(* IEC 61131-3 sources: TA/Tests/RetainTest/OLD/Structure test (part 11) *)

    MATRIX_STRUCTURE_RETAIN.MATRIX_STRING[7,0] := MATRIX_STRUCTURE_RETAIN.MATRIX_STRING[6,0];
    MATRIX_STRUCTURE_RETAIN.MATRIX_STRING[7,1] := MATRIX_STRUCTURE_RETAIN.MATRIX_STRING[6,1];
    MATRIX_STRUCTURE_RETAIN.MATRIX_STRING[7,2] := MATRIX_STRUCTURE_RETAIN.MATRIX_STRING[6,2];
    MATRIX_STRUCTURE_RETAIN.MATRIX_STRING[7,3] := MATRIX_STRUCTURE_RETAIN.MATRIX_STRING[6,3];
    MATRIX_STRUCTURE_RETAIN.MATRIX_STRING[7,4] := MATRIX_STRUCTURE_RETAIN.MATRIX_STRING[6,4];
    MATRIX_STRUCTURE_RETAIN.MATRIX_STRING[7,5] := MATRIX_STRUCTURE_RETAIN.MATRIX_STRING[6,5];
    MATRIX_STRUCTURE_RETAIN.MATRIX_STRING[7,6] := MATRIX_STRUCTURE_RETAIN.MATRIX_STRING[6,6];
    MATRIX_STRUCTURE_RETAIN.MATRIX_STRING[7,7] := MATRIX_STRUCTURE_RETAIN.MATRIX_STRING[6,7];
    MATRIX_STRUCTURE_RETAIN.MATRIX_STRING[7,8] := MATRIX_STRUCTURE_RETAIN.MATRIX_STRING[6,8];
    MATRIX_STRUCTURE_RETAIN.MATRIX_STRING[7,9] := MATRIX_STRUCTURE_RETAIN.MATRIX_STRING[6,9];

    MATRIX_STRUCTURE_RETAIN.MATRIX_TIME[0,0] := MATRIX_STRUCTURE_RETAIN.MATRIX_TIME[0,0] + PULSE_TIME;
    MATRIX_STRUCTURE_RETAIN.MATRIX_TIME[0,1] := MATRIX_STRUCTURE_RETAIN.MATRIX_TIME[0,1] + PULSE_TIME;
    MATRIX_STRUCTURE_RETAIN.MATRIX_TIME[0,2] := MATRIX_STRUCTURE_RETAIN.MATRIX_TIME[0,2] + PULSE_TIME;
    MATRIX_STRUCTURE_RETAIN.MATRIX_TIME[0,3] := MATRIX_STRUCTURE_RETAIN.MATRIX_TIME[0,3] + PULSE_TIME;
    MATRIX_STRUCTURE_RETAIN.MATRIX_TIME[0,4] := MATRIX_STRUCTURE_RETAIN.MATRIX_TIME[0,4] + PULSE_TIME;
    MATRIX_STRUCTURE_RETAIN.MATRIX_TIME[0,5] := MATRIX_STRUCTURE_RETAIN.MATRIX_TIME[0,5] + PULSE_TIME;
    MATRIX_STRUCTURE_RETAIN.MATRIX_TIME[0,6] := MATRIX_STRUCTURE_RETAIN.MATRIX_TIME[0,6] + PULSE_TIME;
    MATRIX_STRUCTURE_RETAIN.MATRIX_TIME[0,7] := MATRIX_STRUCTURE_RETAIN.MATRIX_TIME[0,7] + PULSE_TIME;
    MATRIX_STRUCTURE_RETAIN.MATRIX_TIME[0,8] := MATRIX_STRUCTURE_RETAIN.MATRIX_TIME[0,6];
    MATRIX_STRUCTURE_RETAIN.MATRIX_TIME[0,9] := MATRIX_STRUCTURE_RETAIN.MATRIX_TIME[0,7];

    MATRIX_STRUCTURE_RETAIN.MATRIX_TIME[1,0] := MATRIX_STRUCTURE_RETAIN.MATRIX_TIME[1,0] + PULSE_TIME;
    MATRIX_STRUCTURE_RETAIN.MATRIX_TIME[1,1] := MATRIX_STRUCTURE_RETAIN.MATRIX_TIME[1,1] + PULSE_TIME;
    MATRIX_STRUCTURE_RETAIN.MATRIX_TIME[1,2] := MATRIX_STRUCTURE_RETAIN.MATRIX_TIME[1,2] + PULSE_TIME;
    MATRIX_STRUCTURE_RETAIN.MATRIX_TIME[1,3] := MATRIX_STRUCTURE_RETAIN.MATRIX_TIME[1,3] + PULSE_TIME;
    MATRIX_STRUCTURE_RETAIN.MATRIX_TIME[1,4] := MATRIX_STRUCTURE_RETAIN.MATRIX_TIME[1,4] + PULSE_TIME;
    MATRIX_STRUCTURE_RETAIN.MATRIX_TIME[1,5] := MATRIX_STRUCTURE_RETAIN.MATRIX_TIME[1,5] + PULSE_TIME;
    MATRIX_STRUCTURE_RETAIN.MATRIX_TIME[1,6] := MATRIX_STRUCTURE_RETAIN.MATRIX_TIME[1,6] + PULSE_TIME;
    MATRIX_STRUCTURE_RETAIN.MATRIX_TIME[1,7] := MATRIX_STRUCTURE_RETAIN.MATRIX_TIME[1,7] + PULSE_TIME;
    MATRIX_STRUCTURE_RETAIN.MATRIX_TIME[1,8] := MATRIX_STRUCTURE_RETAIN.MATRIX_TIME[1,6];
    MATRIX_STRUCTURE_RETAIN.MATRIX_TIME[1,9] := MATRIX_STRUCTURE_RETAIN.MATRIX_TIME[1,7];

    MATRIX_STRUCTURE_RETAIN.MATRIX_TIME[2,0] := MATRIX_STRUCTURE_RETAIN.MATRIX_TIME[2,0] + PULSE_TIME;
    MATRIX_STRUCTURE_RETAIN.MATRIX_TIME[2,1] := MATRIX_STRUCTURE_RETAIN.MATRIX_TIME[2,1] + PULSE_TIME;
    MATRIX_STRUCTURE_RETAIN.MATRIX_TIME[2,2] := MATRIX_STRUCTURE_RETAIN.MATRIX_TIME[2,2] + PULSE_TIME;
    MATRIX_STRUCTURE_RETAIN.MATRIX_TIME[2,3] := MATRIX_STRUCTURE_RETAIN.MATRIX_TIME[2,3] + PULSE_TIME;
    MATRIX_STRUCTURE_RETAIN.MATRIX_TIME[2,4] := MATRIX_STRUCTURE_RETAIN.MATRIX_TIME[2,4] + PULSE_TIME;
    MATRIX_STRUCTURE_RETAIN.MATRIX_TIME[2,5] := MATRIX_STRUCTURE_RETAIN.MATRIX_TIME[2,5] + PULSE_TIME;
    MATRIX_STRUCTURE_RETAIN.MATRIX_TIME[2,6] := MATRIX_STRUCTURE_RETAIN.MATRIX_TIME[2,6] + PULSE_TIME;
    MATRIX_STRUCTURE_RETAIN.MATRIX_TIME[2,7] := MATRIX_STRUCTURE_RETAIN.MATRIX_TIME[2,7] + PULSE_TIME;
    MATRIX_STRUCTURE_RETAIN.MATRIX_TIME[2,8] := MATRIX_STRUCTURE_RETAIN.MATRIX_TIME[2,8] + PULSE_TIME;
    MATRIX_STRUCTURE_RETAIN.MATRIX_TIME[2,9] := MATRIX_STRUCTURE_RETAIN.MATRIX_TIME[2,9] + PULSE_TIME;

    MATRIX_STRUCTURE_RETAIN.MATRIX_TIME[3,0] := MATRIX_STRUCTURE_RETAIN.MATRIX_TIME[3,0] + PULSE_TIME;
    MATRIX_STRUCTURE_RETAIN.MATRIX_TIME[3,1] := MATRIX_STRUCTURE_RETAIN.MATRIX_TIME[3,1] + PULSE_TIME;
    MATRIX_STRUCTURE_RETAIN.MATRIX_TIME[3,2] := MATRIX_STRUCTURE_RETAIN.MATRIX_TIME[3,2] + PULSE_TIME;
    MATRIX_STRUCTURE_RETAIN.MATRIX_TIME[3,3] := MATRIX_STRUCTURE_RETAIN.MATRIX_TIME[3,3] + PULSE_TIME;
    MATRIX_STRUCTURE_RETAIN.MATRIX_TIME[3,4] := MATRIX_STRUCTURE_RETAIN.MATRIX_TIME[3,4] + PULSE_TIME;
    MATRIX_STRUCTURE_RETAIN.MATRIX_TIME[3,5] := MATRIX_STRUCTURE_RETAIN.MATRIX_TIME[3,5] + PULSE_TIME;
    MATRIX_STRUCTURE_RETAIN.MATRIX_TIME[3,6] := MATRIX_STRUCTURE_RETAIN.MATRIX_TIME[3,6] + PULSE_TIME;
    MATRIX_STRUCTURE_RETAIN.MATRIX_TIME[3,7] := MATRIX_STRUCTURE_RETAIN.MATRIX_TIME[3,7] + PULSE_TIME;
    MATRIX_STRUCTURE_RETAIN.MATRIX_TIME[3,8] := MATRIX_STRUCTURE_RETAIN.MATRIX_TIME[3,8] + PULSE_TIME;
    MATRIX_STRUCTURE_RETAIN.MATRIX_TIME[3,9] := MATRIX_STRUCTURE_RETAIN.MATRIX_TIME[3,9] + PULSE_TIME;

    MATRIX_STRUCTURE_RETAIN.MATRIX_TIME[4,0] := MATRIX_STRUCTURE_RETAIN.MATRIX_TIME[4,0] + PULSE_TIME;
    MATRIX_STRUCTURE_RETAIN.MATRIX_TIME[4,1] := MATRIX_STRUCTURE_RETAIN.MATRIX_TIME[4,1] + PULSE_TIME;
    MATRIX_STRUCTURE_RETAIN.MATRIX_TIME[4,2] := MATRIX_STRUCTURE_RETAIN.MATRIX_TIME[4,2] + PULSE_TIME;
    MATRIX_STRUCTURE_RETAIN.MATRIX_TIME[4,3] := MATRIX_STRUCTURE_RETAIN.MATRIX_TIME[4,3] + PULSE_TIME;
    MATRIX_STRUCTURE_RETAIN.MATRIX_TIME[4,4] := MATRIX_STRUCTURE_RETAIN.MATRIX_TIME[4,4] + PULSE_TIME;
    MATRIX_STRUCTURE_RETAIN.MATRIX_TIME[4,5] := MATRIX_STRUCTURE_RETAIN.MATRIX_TIME[4,5] + PULSE_TIME;
    MATRIX_STRUCTURE_RETAIN.MATRIX_TIME[4,6] := MATRIX_STRUCTURE_RETAIN.MATRIX_TIME[4,6] + PULSE_TIME;
    MATRIX_STRUCTURE_RETAIN.MATRIX_TIME[4,7] := MATRIX_STRUCTURE_RETAIN.MATRIX_TIME[4,7] + PULSE_TIME;
    MATRIX_STRUCTURE_RETAIN.MATRIX_TIME[4,8] := MATRIX_STRUCTURE_RETAIN.MATRIX_TIME[4,8] + PULSE_TIME;
    MATRIX_STRUCTURE_RETAIN.MATRIX_TIME[4,9] := MATRIX_STRUCTURE_RETAIN.MATRIX_TIME[4,9] + PULSE_TIME;

    MATRIX_STRUCTURE_RETAIN.MATRIX_TIME[5,0] := MATRIX_STRUCTURE_RETAIN.MATRIX_TIME[5,0] + PULSE_TIME;
    MATRIX_STRUCTURE_RETAIN.MATRIX_TIME[5,1] := MATRIX_STRUCTURE_RETAIN.MATRIX_TIME[5,1] + PULSE_TIME;
    MATRIX_STRUCTURE_RETAIN.MATRIX_TIME[5,2] := MATRIX_STRUCTURE_RETAIN.MATRIX_TIME[5,2] + PULSE_TIME;
    MATRIX_STRUCTURE_RETAIN.MATRIX_TIME[5,3] := MATRIX_STRUCTURE_RETAIN.MATRIX_TIME[5,3] + PULSE_TIME;
    MATRIX_STRUCTURE_RETAIN.MATRIX_TIME[5,4] := MATRIX_STRUCTURE_RETAIN.MATRIX_TIME[5,4] + PULSE_TIME;
    MATRIX_STRUCTURE_RETAIN.MATRIX_TIME[5,5] := MATRIX_STRUCTURE_RETAIN.MATRIX_TIME[5,5] + PULSE_TIME;
    MATRIX_STRUCTURE_RETAIN.MATRIX_TIME[5,6] := MATRIX_STRUCTURE_RETAIN.MATRIX_TIME[5,6] + PULSE_TIME;
    MATRIX_STRUCTURE_RETAIN.MATRIX_TIME[5,7] := MATRIX_STRUCTURE_RETAIN.MATRIX_TIME[5,7] + PULSE_TIME;
    MATRIX_STRUCTURE_RETAIN.MATRIX_TIME[5,8] := MATRIX_STRUCTURE_RETAIN.MATRIX_TIME[5,8] + PULSE_TIME;
    MATRIX_STRUCTURE_RETAIN.MATRIX_TIME[5,9] := MATRIX_STRUCTURE_RETAIN.MATRIX_TIME[5,9] + PULSE_TIME;

    MATRIX_STRUCTURE_RETAIN.MATRIX_TIME[6,0] := MATRIX_STRUCTURE_RETAIN.MATRIX_TIME[6,0] + PULSE_TIME;
    MATRIX_STRUCTURE_RETAIN.MATRIX_TIME[6,1] := MATRIX_STRUCTURE_RETAIN.MATRIX_TIME[6,1] + PULSE_TIME;
    MATRIX_STRUCTURE_RETAIN.MATRIX_TIME[6,2] := MATRIX_STRUCTURE_RETAIN.MATRIX_TIME[6,2] + PULSE_TIME;
    MATRIX_STRUCTURE_RETAIN.MATRIX_TIME[6,3] := MATRIX_STRUCTURE_RETAIN.MATRIX_TIME[6,3] + PULSE_TIME;
    MATRIX_STRUCTURE_RETAIN.MATRIX_TIME[6,4] := MATRIX_STRUCTURE_RETAIN.MATRIX_TIME[6,4] + PULSE_TIME;
    MATRIX_STRUCTURE_RETAIN.MATRIX_TIME[6,5] := MATRIX_STRUCTURE_RETAIN.MATRIX_TIME[6,5] + PULSE_TIME;
    MATRIX_STRUCTURE_RETAIN.MATRIX_TIME[6,6] := MATRIX_STRUCTURE_RETAIN.MATRIX_TIME[6,6] + PULSE_TIME;
    MATRIX_STRUCTURE_RETAIN.MATRIX_TIME[6,7] := MATRIX_STRUCTURE_RETAIN.MATRIX_TIME[6,7] + PULSE_TIME;
    MATRIX_STRUCTURE_RETAIN.MATRIX_TIME[6,8] := MATRIX_STRUCTURE_RETAIN.MATRIX_TIME[6,8] + PULSE_TIME;
    MATRIX_STRUCTURE_RETAIN.MATRIX_TIME[6,9] := MATRIX_STRUCTURE_RETAIN.MATRIX_TIME[6,9] + PULSE_TIME;

    MATRIX_STRUCTURE_RETAIN.MATRIX_TIME[7,0] := MATRIX_STRUCTURE_RETAIN.MATRIX_TIME[6,0];
    MATRIX_STRUCTURE_RETAIN.MATRIX_TIME[7,1] := MATRIX_STRUCTURE_RETAIN.MATRIX_TIME[6,1];
    MATRIX_STRUCTURE_RETAIN.MATRIX_TIME[7,2] := MATRIX_STRUCTURE_RETAIN.MATRIX_TIME[6,2];
    MATRIX_STRUCTURE_RETAIN.MATRIX_TIME[7,3] := MATRIX_STRUCTURE_RETAIN.MATRIX_TIME[6,3];
    MATRIX_STRUCTURE_RETAIN.MATRIX_TIME[7,4] := MATRIX_STRUCTURE_RETAIN.MATRIX_TIME[6,4];
    MATRIX_STRUCTURE_RETAIN.MATRIX_TIME[7,5] := MATRIX_STRUCTURE_RETAIN.MATRIX_TIME[6,5];
    MATRIX_STRUCTURE_RETAIN.MATRIX_TIME[7,6] := MATRIX_STRUCTURE_RETAIN.MATRIX_TIME[6,6];
    MATRIX_STRUCTURE_RETAIN.MATRIX_TIME[7,7] := MATRIX_STRUCTURE_RETAIN.MATRIX_TIME[6,7];
    MATRIX_STRUCTURE_RETAIN.MATRIX_TIME[7,8] := MATRIX_STRUCTURE_RETAIN.MATRIX_TIME[6,6];
    MATRIX_STRUCTURE_RETAIN.MATRIX_TIME[7,9] := MATRIX_STRUCTURE_RETAIN.MATRIX_TIME[6,7];

    MATRIX_STRUCTURE_RETAIN.MATRIX_UDINT[0,0] := MATRIX_STRUCTURE_RETAIN.MATRIX_UDINT[0,0] + 1;
    MATRIX_STRUCTURE_RETAIN.MATRIX_UDINT[0,1] := MATRIX_STRUCTURE_RETAIN.MATRIX_UDINT[0,1] + 1;
    MATRIX_STRUCTURE_RETAIN.MATRIX_UDINT[0,2] := MATRIX_STRUCTURE_RETAIN.MATRIX_UDINT[0,2] + 1;
    MATRIX_STRUCTURE_RETAIN.MATRIX_UDINT[0,3] := MATRIX_STRUCTURE_RETAIN.MATRIX_UDINT[0,3] + 1;
    MATRIX_STRUCTURE_RETAIN.MATRIX_UDINT[0,4] := MATRIX_STRUCTURE_RETAIN.MATRIX_UDINT[0,4] + 1;
    MATRIX_STRUCTURE_RETAIN.MATRIX_UDINT[0,5] := MATRIX_STRUCTURE_RETAIN.MATRIX_UDINT[0,5] + 1;
    MATRIX_STRUCTURE_RETAIN.MATRIX_UDINT[0,6] := MATRIX_STRUCTURE_RETAIN.MATRIX_UDINT[0,6] + 1;
    MATRIX_STRUCTURE_RETAIN.MATRIX_UDINT[0,7] := MATRIX_STRUCTURE_RETAIN.MATRIX_UDINT[0,7] + 1;
    MATRIX_STRUCTURE_RETAIN.MATRIX_UDINT[0,8] := MATRIX_STRUCTURE_RETAIN.MATRIX_UDINT[0,6];
    MATRIX_STRUCTURE_RETAIN.MATRIX_UDINT[0,9] := MATRIX_STRUCTURE_RETAIN.MATRIX_UDINT[0,7];

    MATRIX_STRUCTURE_RETAIN.MATRIX_UDINT[1,0] := MATRIX_STRUCTURE_RETAIN.MATRIX_UDINT[1,0] + 1;
    MATRIX_STRUCTURE_RETAIN.MATRIX_UDINT[1,1] := MATRIX_STRUCTURE_RETAIN.MATRIX_UDINT[1,1] + 1;
    MATRIX_STRUCTURE_RETAIN.MATRIX_UDINT[1,2] := MATRIX_STRUCTURE_RETAIN.MATRIX_UDINT[1,2] + 1;
    MATRIX_STRUCTURE_RETAIN.MATRIX_UDINT[1,3] := MATRIX_STRUCTURE_RETAIN.MATRIX_UDINT[1,3] + 1;
    MATRIX_STRUCTURE_RETAIN.MATRIX_UDINT[1,4] := MATRIX_STRUCTURE_RETAIN.MATRIX_UDINT[1,4] + 1;
    MATRIX_STRUCTURE_RETAIN.MATRIX_UDINT[1,5] := MATRIX_STRUCTURE_RETAIN.MATRIX_UDINT[1,5] + 1;
    MATRIX_STRUCTURE_RETAIN.MATRIX_UDINT[1,6] := MATRIX_STRUCTURE_RETAIN.MATRIX_UDINT[1,6] + 1;
    MATRIX_STRUCTURE_RETAIN.MATRIX_UDINT[1,7] := MATRIX_STRUCTURE_RETAIN.MATRIX_UDINT[1,7] + 1;
    MATRIX_STRUCTURE_RETAIN.MATRIX_UDINT[1,8] := MATRIX_STRUCTURE_RETAIN.MATRIX_UDINT[1,6];
    MATRIX_STRUCTURE_RETAIN.MATRIX_UDINT[1,9] := MATRIX_STRUCTURE_RETAIN.MATRIX_UDINT[1,7];

    MATRIX_STRUCTURE_RETAIN.MATRIX_UDINT[2,0] := MATRIX_STRUCTURE_RETAIN.MATRIX_UDINT[2,0] + 1;
    MATRIX_STRUCTURE_RETAIN.MATRIX_UDINT[2,1] := MATRIX_STRUCTURE_RETAIN.MATRIX_UDINT[2,1] + 1;
    MATRIX_STRUCTURE_RETAIN.MATRIX_UDINT[2,2] := MATRIX_STRUCTURE_RETAIN.MATRIX_UDINT[2,2] + 1;
    MATRIX_STRUCTURE_RETAIN.MATRIX_UDINT[2,3] := MATRIX_STRUCTURE_RETAIN.MATRIX_UDINT[2,3] + 1;
    MATRIX_STRUCTURE_RETAIN.MATRIX_UDINT[2,4] := MATRIX_STRUCTURE_RETAIN.MATRIX_UDINT[2,4] + 1;
    MATRIX_STRUCTURE_RETAIN.MATRIX_UDINT[2,5] := MATRIX_STRUCTURE_RETAIN.MATRIX_UDINT[2,5] + 1;
    MATRIX_STRUCTURE_RETAIN.MATRIX_UDINT[2,6] := MATRIX_STRUCTURE_RETAIN.MATRIX_UDINT[2,6] + 1;
    MATRIX_STRUCTURE_RETAIN.MATRIX_UDINT[2,7] := MATRIX_STRUCTURE_RETAIN.MATRIX_UDINT[2,7] + 1;
    MATRIX_STRUCTURE_RETAIN.MATRIX_UDINT[2,8] := MATRIX_STRUCTURE_RETAIN.MATRIX_UDINT[2,8] + 1;
    MATRIX_STRUCTURE_RETAIN.MATRIX_UDINT[2,9] := MATRIX_STRUCTURE_RETAIN.MATRIX_UDINT[2,9] + 1;

    MATRIX_STRUCTURE_RETAIN.MATRIX_UDINT[3,0] := MATRIX_STRUCTURE_RETAIN.MATRIX_UDINT[3,0] + 1;
    MATRIX_STRUCTURE_RETAIN.MATRIX_UDINT[3,1] := MATRIX_STRUCTURE_RETAIN.MATRIX_UDINT[3,1] + 1;
    MATRIX_STRUCTURE_RETAIN.MATRIX_UDINT[3,2] := MATRIX_STRUCTURE_RETAIN.MATRIX_UDINT[3,2] + 1;
    MATRIX_STRUCTURE_RETAIN.MATRIX_UDINT[3,3] := MATRIX_STRUCTURE_RETAIN.MATRIX_UDINT[3,3] + 1;
    MATRIX_STRUCTURE_RETAIN.MATRIX_UDINT[3,4] := MATRIX_STRUCTURE_RETAIN.MATRIX_UDINT[3,4] + 1;
    MATRIX_STRUCTURE_RETAIN.MATRIX_UDINT[3,5] := MATRIX_STRUCTURE_RETAIN.MATRIX_UDINT[3,5] + 1;
    MATRIX_STRUCTURE_RETAIN.MATRIX_UDINT[3,6] := MATRIX_STRUCTURE_RETAIN.MATRIX_UDINT[3,6] + 1;
    MATRIX_STRUCTURE_RETAIN.MATRIX_UDINT[3,7] := MATRIX_STRUCTURE_RETAIN.MATRIX_UDINT[3,7] + 1;
    MATRIX_STRUCTURE_RETAIN.MATRIX_UDINT[3,8] := MATRIX_STRUCTURE_RETAIN.MATRIX_UDINT[3,8] + 1;
    MATRIX_STRUCTURE_RETAIN.MATRIX_UDINT[3,9] := MATRIX_STRUCTURE_RETAIN.MATRIX_UDINT[3,9] + 1;

    MATRIX_STRUCTURE_RETAIN.MATRIX_UDINT[4,0] := MATRIX_STRUCTURE_RETAIN.MATRIX_UDINT[4,0] + 1;
    MATRIX_STRUCTURE_RETAIN.MATRIX_UDINT[4,1] := MATRIX_STRUCTURE_RETAIN.MATRIX_UDINT[4,1] + 1;
    MATRIX_STRUCTURE_RETAIN.MATRIX_UDINT[4,2] := MATRIX_STRUCTURE_RETAIN.MATRIX_UDINT[4,2] + 1;
    MATRIX_STRUCTURE_RETAIN.MATRIX_UDINT[4,3] := MATRIX_STRUCTURE_RETAIN.MATRIX_UDINT[4,3] + 1;
    MATRIX_STRUCTURE_RETAIN.MATRIX_UDINT[4,4] := MATRIX_STRUCTURE_RETAIN.MATRIX_UDINT[4,4] + 1;
    MATRIX_STRUCTURE_RETAIN.MATRIX_UDINT[4,5] := MATRIX_STRUCTURE_RETAIN.MATRIX_UDINT[4,5] + 1;
    MATRIX_STRUCTURE_RETAIN.MATRIX_UDINT[4,6] := MATRIX_STRUCTURE_RETAIN.MATRIX_UDINT[4,6] + 1;
    MATRIX_STRUCTURE_RETAIN.MATRIX_UDINT[4,7] := MATRIX_STRUCTURE_RETAIN.MATRIX_UDINT[4,7] + 1;
    MATRIX_STRUCTURE_RETAIN.MATRIX_UDINT[4,8] := MATRIX_STRUCTURE_RETAIN.MATRIX_UDINT[4,8] + 1;
    MATRIX_STRUCTURE_RETAIN.MATRIX_UDINT[4,9] := MATRIX_STRUCTURE_RETAIN.MATRIX_UDINT[4,9] + 1;

    MATRIX_STRUCTURE_RETAIN.MATRIX_UDINT[5,0] := MATRIX_STRUCTURE_RETAIN.MATRIX_UDINT[5,0] + 1;
    MATRIX_STRUCTURE_RETAIN.MATRIX_UDINT[5,1] := MATRIX_STRUCTURE_RETAIN.MATRIX_UDINT[5,1] + 1;
    MATRIX_STRUCTURE_RETAIN.MATRIX_UDINT[5,2] := MATRIX_STRUCTURE_RETAIN.MATRIX_UDINT[5,2] + 1;
    MATRIX_STRUCTURE_RETAIN.MATRIX_UDINT[5,3] := MATRIX_STRUCTURE_RETAIN.MATRIX_UDINT[5,3] + 1;
    MATRIX_STRUCTURE_RETAIN.MATRIX_UDINT[5,4] := MATRIX_STRUCTURE_RETAIN.MATRIX_UDINT[5,4] + 1;
    MATRIX_STRUCTURE_RETAIN.MATRIX_UDINT[5,5] := MATRIX_STRUCTURE_RETAIN.MATRIX_UDINT[5,5] + 1;
    MATRIX_STRUCTURE_RETAIN.MATRIX_UDINT[5,6] := MATRIX_STRUCTURE_RETAIN.MATRIX_UDINT[5,6] + 1;
    MATRIX_STRUCTURE_RETAIN.MATRIX_UDINT[5,7] := MATRIX_STRUCTURE_RETAIN.MATRIX_UDINT[5,7] + 1;
    MATRIX_STRUCTURE_RETAIN.MATRIX_UDINT[5,8] := MATRIX_STRUCTURE_RETAIN.MATRIX_UDINT[5,8] + 1;
    MATRIX_STRUCTURE_RETAIN.MATRIX_UDINT[5,9] := MATRIX_STRUCTURE_RETAIN.MATRIX_UDINT[5,9] + 1;

    MATRIX_STRUCTURE_RETAIN.MATRIX_UDINT[6,0] := MATRIX_STRUCTURE_RETAIN.MATRIX_UDINT[6,0] + 1;
    MATRIX_STRUCTURE_RETAIN.MATRIX_UDINT[6,1] := MATRIX_STRUCTURE_RETAIN.MATRIX_UDINT[6,1] + 1;
    MATRIX_STRUCTURE_RETAIN.MATRIX_UDINT[6,2] := MATRIX_STRUCTURE_RETAIN.MATRIX_UDINT[6,2] + 1;
    MATRIX_STRUCTURE_RETAIN.MATRIX_UDINT[6,3] := MATRIX_STRUCTURE_RETAIN.MATRIX_UDINT[6,3] + 1;
    MATRIX_STRUCTURE_RETAIN.MATRIX_UDINT[6,4] := MATRIX_STRUCTURE_RETAIN.MATRIX_UDINT[6,4] + 1;
    MATRIX_STRUCTURE_RETAIN.MATRIX_UDINT[6,5] := MATRIX_STRUCTURE_RETAIN.MATRIX_UDINT[6,5] + 1;
    MATRIX_STRUCTURE_RETAIN.MATRIX_UDINT[6,6] := MATRIX_STRUCTURE_RETAIN.MATRIX_UDINT[6,6] + 1;
    MATRIX_STRUCTURE_RETAIN.MATRIX_UDINT[6,7] := MATRIX_STRUCTURE_RETAIN.MATRIX_UDINT[6,7] + 1;
    MATRIX_STRUCTURE_RETAIN.MATRIX_UDINT[6,8] := MATRIX_STRUCTURE_RETAIN.MATRIX_UDINT[6,8] + 1;
    MATRIX_STRUCTURE_RETAIN.MATRIX_UDINT[6,9] := MATRIX_STRUCTURE_RETAIN.MATRIX_UDINT[6,9] + 1;

    MATRIX_STRUCTURE_RETAIN.MATRIX_UDINT[7,0] := MATRIX_STRUCTURE_RETAIN.MATRIX_UDINT[6,0];
    MATRIX_STRUCTURE_RETAIN.MATRIX_UDINT[7,1] := MATRIX_STRUCTURE_RETAIN.MATRIX_UDINT[6,1];
    MATRIX_STRUCTURE_RETAIN.MATRIX_UDINT[7,2] := MATRIX_STRUCTURE_RETAIN.MATRIX_UDINT[6,2];
    MATRIX_STRUCTURE_RETAIN.MATRIX_UDINT[7,3] := MATRIX_STRUCTURE_RETAIN.MATRIX_UDINT[6,3];
    MATRIX_STRUCTURE_RETAIN.MATRIX_UDINT[7,4] := MATRIX_STRUCTURE_RETAIN.MATRIX_UDINT[6,4];
    MATRIX_STRUCTURE_RETAIN.MATRIX_UDINT[7,5] := MATRIX_STRUCTURE_RETAIN.MATRIX_UDINT[6,5];
    MATRIX_STRUCTURE_RETAIN.MATRIX_UDINT[7,6] := MATRIX_STRUCTURE_RETAIN.MATRIX_UDINT[6,6];
    MATRIX_STRUCTURE_RETAIN.MATRIX_UDINT[7,7] := MATRIX_STRUCTURE_RETAIN.MATRIX_UDINT[6,7];
    MATRIX_STRUCTURE_RETAIN.MATRIX_UDINT[7,8] := MATRIX_STRUCTURE_RETAIN.MATRIX_UDINT[6,8];
    MATRIX_STRUCTURE_RETAIN.MATRIX_UDINT[7,9] := MATRIX_STRUCTURE_RETAIN.MATRIX_UDINT[6,9];

    MATRIX_STRUCTURE_RETAIN.MATRIX_UINT[0,0] := MATRIX_STRUCTURE_RETAIN.MATRIX_UINT[0,0] + 1;
    MATRIX_STRUCTURE_RETAIN.MATRIX_UINT[0,1] := MATRIX_STRUCTURE_RETAIN.MATRIX_UINT[0,1] + 1;
    MATRIX_STRUCTURE_RETAIN.MATRIX_UINT[0,2] := MATRIX_STRUCTURE_RETAIN.MATRIX_UINT[0,2] + 1;
    MATRIX_STRUCTURE_RETAIN.MATRIX_UINT[0,3] := MATRIX_STRUCTURE_RETAIN.MATRIX_UINT[0,3] + 1;
    MATRIX_STRUCTURE_RETAIN.MATRIX_UINT[0,4] := MATRIX_STRUCTURE_RETAIN.MATRIX_UINT[0,4] + 1;
    MATRIX_STRUCTURE_RETAIN.MATRIX_UINT[0,5] := MATRIX_STRUCTURE_RETAIN.MATRIX_UINT[0,5] + 1;
    MATRIX_STRUCTURE_RETAIN.MATRIX_UINT[0,6] := MATRIX_STRUCTURE_RETAIN.MATRIX_UINT[0,6] + 1;
    MATRIX_STRUCTURE_RETAIN.MATRIX_UINT[0,7] := MATRIX_STRUCTURE_RETAIN.MATRIX_UINT[0,7] + 1;
    MATRIX_STRUCTURE_RETAIN.MATRIX_UINT[0,8] := MATRIX_STRUCTURE_RETAIN.MATRIX_UINT[0,6];
    MATRIX_STRUCTURE_RETAIN.MATRIX_UINT[0,9] := MATRIX_STRUCTURE_RETAIN.MATRIX_UINT[0,7];

    MATRIX_STRUCTURE_RETAIN.MATRIX_UINT[1,0] := MATRIX_STRUCTURE_RETAIN.MATRIX_UINT[1,0] + 1;
    MATRIX_STRUCTURE_RETAIN.MATRIX_UINT[1,1] := MATRIX_STRUCTURE_RETAIN.MATRIX_UINT[1,1] + 1;
    MATRIX_STRUCTURE_RETAIN.MATRIX_UINT[1,2] := MATRIX_STRUCTURE_RETAIN.MATRIX_UINT[1,2] + 1;
    MATRIX_STRUCTURE_RETAIN.MATRIX_UINT[1,3] := MATRIX_STRUCTURE_RETAIN.MATRIX_UINT[1,3] + 1;
    MATRIX_STRUCTURE_RETAIN.MATRIX_UINT[1,4] := MATRIX_STRUCTURE_RETAIN.MATRIX_UINT[1,4] + 1;
    MATRIX_STRUCTURE_RETAIN.MATRIX_UINT[1,5] := MATRIX_STRUCTURE_RETAIN.MATRIX_UINT[1,5] + 1;
    MATRIX_STRUCTURE_RETAIN.MATRIX_UINT[1,6] := MATRIX_STRUCTURE_RETAIN.MATRIX_UINT[1,6] + 1;
    MATRIX_STRUCTURE_RETAIN.MATRIX_UINT[1,7] := MATRIX_STRUCTURE_RETAIN.MATRIX_UINT[1,7] + 1;
    MATRIX_STRUCTURE_RETAIN.MATRIX_UINT[1,8] := MATRIX_STRUCTURE_RETAIN.MATRIX_UINT[1,6];
    MATRIX_STRUCTURE_RETAIN.MATRIX_UINT[1,9] := MATRIX_STRUCTURE_RETAIN.MATRIX_UINT[1,7];

    MATRIX_STRUCTURE_RETAIN.MATRIX_UINT[2,0] := MATRIX_STRUCTURE_RETAIN.MATRIX_UINT[2,0] + 1;
    MATRIX_STRUCTURE_RETAIN.MATRIX_UINT[2,1] := MATRIX_STRUCTURE_RETAIN.MATRIX_UINT[2,1] + 1;
    MATRIX_STRUCTURE_RETAIN.MATRIX_UINT[2,2] := MATRIX_STRUCTURE_RETAIN.MATRIX_UINT[2,2] + 1;
    MATRIX_STRUCTURE_RETAIN.MATRIX_UINT[2,3] := MATRIX_STRUCTURE_RETAIN.MATRIX_UINT[2,3] + 1;
    MATRIX_STRUCTURE_RETAIN.MATRIX_UINT[2,4] := MATRIX_STRUCTURE_RETAIN.MATRIX_UINT[2,4] + 1;
    MATRIX_STRUCTURE_RETAIN.MATRIX_UINT[2,5] := MATRIX_STRUCTURE_RETAIN.MATRIX_UINT[2,5] + 1;
    MATRIX_STRUCTURE_RETAIN.MATRIX_UINT[2,6] := MATRIX_STRUCTURE_RETAIN.MATRIX_UINT[2,6] + 1;
    MATRIX_STRUCTURE_RETAIN.MATRIX_UINT[2,7] := MATRIX_STRUCTURE_RETAIN.MATRIX_UINT[2,7] + 1;
    MATRIX_STRUCTURE_RETAIN.MATRIX_UINT[2,8] := MATRIX_STRUCTURE_RETAIN.MATRIX_UINT[2,8] + 1;
    MATRIX_STRUCTURE_RETAIN.MATRIX_UINT[2,9] := MATRIX_STRUCTURE_RETAIN.MATRIX_UINT[2,9] + 1;

    MATRIX_STRUCTURE_RETAIN.MATRIX_UINT[3,0] := MATRIX_STRUCTURE_RETAIN.MATRIX_UINT[3,0] + 1;
    MATRIX_STRUCTURE_RETAIN.MATRIX_UINT[3,1] := MATRIX_STRUCTURE_RETAIN.MATRIX_UINT[3,1] + 1;
    MATRIX_STRUCTURE_RETAIN.MATRIX_UINT[3,2] := MATRIX_STRUCTURE_RETAIN.MATRIX_UINT[3,2] + 1;
    MATRIX_STRUCTURE_RETAIN.MATRIX_UINT[3,3] := MATRIX_STRUCTURE_RETAIN.MATRIX_UINT[3,3] + 1;
    MATRIX_STRUCTURE_RETAIN.MATRIX_UINT[3,4] := MATRIX_STRUCTURE_RETAIN.MATRIX_UINT[3,4] + 1;
    MATRIX_STRUCTURE_RETAIN.MATRIX_UINT[3,5] := MATRIX_STRUCTURE_RETAIN.MATRIX_UINT[3,5] + 1;
    MATRIX_STRUCTURE_RETAIN.MATRIX_UINT[3,6] := MATRIX_STRUCTURE_RETAIN.MATRIX_UINT[3,6] + 1;
    MATRIX_STRUCTURE_RETAIN.MATRIX_UINT[3,7] := MATRIX_STRUCTURE_RETAIN.MATRIX_UINT[3,7] + 1;
    MATRIX_STRUCTURE_RETAIN.MATRIX_UINT[3,8] := MATRIX_STRUCTURE_RETAIN.MATRIX_UINT[3,8] + 1;
    MATRIX_STRUCTURE_RETAIN.MATRIX_UINT[3,9] := MATRIX_STRUCTURE_RETAIN.MATRIX_UINT[3,9] + 1;

    MATRIX_STRUCTURE_RETAIN.MATRIX_UINT[4,0] := MATRIX_STRUCTURE_RETAIN.MATRIX_UINT[4,0] + 1;
    MATRIX_STRUCTURE_RETAIN.MATRIX_UINT[4,1] := MATRIX_STRUCTURE_RETAIN.MATRIX_UINT[4,1] + 1;
    MATRIX_STRUCTURE_RETAIN.MATRIX_UINT[4,2] := MATRIX_STRUCTURE_RETAIN.MATRIX_UINT[4,2] + 1;
    MATRIX_STRUCTURE_RETAIN.MATRIX_UINT[4,3] := MATRIX_STRUCTURE_RETAIN.MATRIX_UINT[4,3] + 1;
    MATRIX_STRUCTURE_RETAIN.MATRIX_UINT[4,4] := MATRIX_STRUCTURE_RETAIN.MATRIX_UINT[4,4] + 1;
    MATRIX_STRUCTURE_RETAIN.MATRIX_UINT[4,5] := MATRIX_STRUCTURE_RETAIN.MATRIX_UINT[4,5] + 1;
    MATRIX_STRUCTURE_RETAIN.MATRIX_UINT[4,6] := MATRIX_STRUCTURE_RETAIN.MATRIX_UINT[4,6] + 1;
    MATRIX_STRUCTURE_RETAIN.MATRIX_UINT[4,7] := MATRIX_STRUCTURE_RETAIN.MATRIX_UINT[4,7] + 1;
    MATRIX_STRUCTURE_RETAIN.MATRIX_UINT[4,8] := MATRIX_STRUCTURE_RETAIN.MATRIX_UINT[4,8] + 1;
    MATRIX_STRUCTURE_RETAIN.MATRIX_UINT[4,9] := MATRIX_STRUCTURE_RETAIN.MATRIX_UINT[4,9] + 1;

    MATRIX_STRUCTURE_RETAIN.MATRIX_UINT[5,0] := MATRIX_STRUCTURE_RETAIN.MATRIX_UINT[5,0] + 1;
    MATRIX_STRUCTURE_RETAIN.MATRIX_UINT[5,1] := MATRIX_STRUCTURE_RETAIN.MATRIX_UINT[5,1] + 1;
    MATRIX_STRUCTURE_RETAIN.MATRIX_UINT[5,2] := MATRIX_STRUCTURE_RETAIN.MATRIX_UINT[5,2] + 1;
    MATRIX_STRUCTURE_RETAIN.MATRIX_UINT[5,3] := MATRIX_STRUCTURE_RETAIN.MATRIX_UINT[5,3] + 1;
    MATRIX_STRUCTURE_RETAIN.MATRIX_UINT[5,4] := MATRIX_STRUCTURE_RETAIN.MATRIX_UINT[5,4] + 1;
    MATRIX_STRUCTURE_RETAIN.MATRIX_UINT[5,5] := MATRIX_STRUCTURE_RETAIN.MATRIX_UINT[5,5] + 1;
    MATRIX_STRUCTURE_RETAIN.MATRIX_UINT[5,6] := MATRIX_STRUCTURE_RETAIN.MATRIX_UINT[5,6] + 1;
    MATRIX_STRUCTURE_RETAIN.MATRIX_UINT[5,7] := MATRIX_STRUCTURE_RETAIN.MATRIX_UINT[5,7] + 1;
    MATRIX_STRUCTURE_RETAIN.MATRIX_UINT[5,8] := MATRIX_STRUCTURE_RETAIN.MATRIX_UINT[5,8] + 1;
    MATRIX_STRUCTURE_RETAIN.MATRIX_UINT[5,9] := MATRIX_STRUCTURE_RETAIN.MATRIX_UINT[5,9] + 1;

    MATRIX_STRUCTURE_RETAIN.MATRIX_UINT[6,0] := MATRIX_STRUCTURE_RETAIN.MATRIX_UINT[6,0] + 1;
    MATRIX_STRUCTURE_RETAIN.MATRIX_UINT[6,1] := MATRIX_STRUCTURE_RETAIN.MATRIX_UINT[6,1] + 1;
    MATRIX_STRUCTURE_RETAIN.MATRIX_UINT[6,2] := MATRIX_STRUCTURE_RETAIN.MATRIX_UINT[6,2] + 1;
    MATRIX_STRUCTURE_RETAIN.MATRIX_UINT[6,3] := MATRIX_STRUCTURE_RETAIN.MATRIX_UINT[6,3] + 1;
    MATRIX_STRUCTURE_RETAIN.MATRIX_UINT[6,4] := MATRIX_STRUCTURE_RETAIN.MATRIX_UINT[6,4] + 1;
    MATRIX_STRUCTURE_RETAIN.MATRIX_UINT[6,5] := MATRIX_STRUCTURE_RETAIN.MATRIX_UINT[6,5] + 1;
    MATRIX_STRUCTURE_RETAIN.MATRIX_UINT[6,6] := MATRIX_STRUCTURE_RETAIN.MATRIX_UINT[6,6] + 1;
    MATRIX_STRUCTURE_RETAIN.MATRIX_UINT[6,7] := MATRIX_STRUCTURE_RETAIN.MATRIX_UINT[6,7] + 1;
    MATRIX_STRUCTURE_RETAIN.MATRIX_UINT[6,8] := MATRIX_STRUCTURE_RETAIN.MATRIX_UINT[6,8] + 1;
    MATRIX_STRUCTURE_RETAIN.MATRIX_UINT[6,9] := MATRIX_STRUCTURE_RETAIN.MATRIX_UINT[6,9] + 1;

    MATRIX_STRUCTURE_RETAIN.MATRIX_UINT[7,0] := MATRIX_STRUCTURE_RETAIN.MATRIX_UINT[6,0];
    MATRIX_STRUCTURE_RETAIN.MATRIX_UINT[7,1] := MATRIX_STRUCTURE_RETAIN.MATRIX_UINT[6,1];
    MATRIX_STRUCTURE_RETAIN.MATRIX_UINT[7,2] := MATRIX_STRUCTURE_RETAIN.MATRIX_UINT[6,2];
    MATRIX_STRUCTURE_RETAIN.MATRIX_UINT[7,3] := MATRIX_STRUCTURE_RETAIN.MATRIX_UINT[6,3];
    MATRIX_STRUCTURE_RETAIN.MATRIX_UINT[7,4] := MATRIX_STRUCTURE_RETAIN.MATRIX_UINT[6,4];
    MATRIX_STRUCTURE_RETAIN.MATRIX_UINT[7,5] := MATRIX_STRUCTURE_RETAIN.MATRIX_UINT[6,5];
    MATRIX_STRUCTURE_RETAIN.MATRIX_UINT[7,6] := MATRIX_STRUCTURE_RETAIN.MATRIX_UINT[6,6];
    MATRIX_STRUCTURE_RETAIN.MATRIX_UINT[7,7] := MATRIX_STRUCTURE_RETAIN.MATRIX_UINT[6,7];
    MATRIX_STRUCTURE_RETAIN.MATRIX_UINT[7,8] := MATRIX_STRUCTURE_RETAIN.MATRIX_UINT[6,8];
    MATRIX_STRUCTURE_RETAIN.MATRIX_UINT[7,9] := MATRIX_STRUCTURE_RETAIN.MATRIX_UINT[6,9];

    MATRIX_STRUCTURE_RETAIN.MATRIX_ULINT[0,0] := MATRIX_STRUCTURE_RETAIN.MATRIX_ULINT[0,0] + 1;
    MATRIX_STRUCTURE_RETAIN.MATRIX_ULINT[0,1] := MATRIX_STRUCTURE_RETAIN.MATRIX_ULINT[0,1] + 1;
    MATRIX_STRUCTURE_RETAIN.MATRIX_ULINT[0,2] := MATRIX_STRUCTURE_RETAIN.MATRIX_ULINT[0,2] + 1;
    MATRIX_STRUCTURE_RETAIN.MATRIX_ULINT[0,3] := MATRIX_STRUCTURE_RETAIN.MATRIX_ULINT[0,3] + 1;
    MATRIX_STRUCTURE_RETAIN.MATRIX_ULINT[0,4] := MATRIX_STRUCTURE_RETAIN.MATRIX_ULINT[0,4] + 1;
    MATRIX_STRUCTURE_RETAIN.MATRIX_ULINT[0,5] := MATRIX_STRUCTURE_RETAIN.MATRIX_ULINT[0,5] + 1;
    MATRIX_STRUCTURE_RETAIN.MATRIX_ULINT[0,6] := MATRIX_STRUCTURE_RETAIN.MATRIX_ULINT[0,6] + 1;
    MATRIX_STRUCTURE_RETAIN.MATRIX_ULINT[0,7] := MATRIX_STRUCTURE_RETAIN.MATRIX_ULINT[0,7] + 1;
    MATRIX_STRUCTURE_RETAIN.MATRIX_ULINT[0,8] := MATRIX_STRUCTURE_RETAIN.MATRIX_ULINT[0,6];
    MATRIX_STRUCTURE_RETAIN.MATRIX_ULINT[0,9] := MATRIX_STRUCTURE_RETAIN.MATRIX_ULINT[0,7];

    MATRIX_STRUCTURE_RETAIN.MATRIX_ULINT[1,0] := MATRIX_STRUCTURE_RETAIN.MATRIX_ULINT[1,0] + 1;
    MATRIX_STRUCTURE_RETAIN.MATRIX_ULINT[1,1] := MATRIX_STRUCTURE_RETAIN.MATRIX_ULINT[1,1] + 1;
    MATRIX_STRUCTURE_RETAIN.MATRIX_ULINT[1,2] := MATRIX_STRUCTURE_RETAIN.MATRIX_ULINT[1,2] + 1;
    MATRIX_STRUCTURE_RETAIN.MATRIX_ULINT[1,3] := MATRIX_STRUCTURE_RETAIN.MATRIX_ULINT[1,3] + 1;
    MATRIX_STRUCTURE_RETAIN.MATRIX_ULINT[1,4] := MATRIX_STRUCTURE_RETAIN.MATRIX_ULINT[1,4] + 1;
    MATRIX_STRUCTURE_RETAIN.MATRIX_ULINT[1,5] := MATRIX_STRUCTURE_RETAIN.MATRIX_ULINT[1,5] + 1;
    MATRIX_STRUCTURE_RETAIN.MATRIX_ULINT[1,6] := MATRIX_STRUCTURE_RETAIN.MATRIX_ULINT[1,6] + 1;
    MATRIX_STRUCTURE_RETAIN.MATRIX_ULINT[1,7] := MATRIX_STRUCTURE_RETAIN.MATRIX_ULINT[1,7] + 1;
    MATRIX_STRUCTURE_RETAIN.MATRIX_ULINT[1,8] := MATRIX_STRUCTURE_RETAIN.MATRIX_ULINT[1,6];
    MATRIX_STRUCTURE_RETAIN.MATRIX_ULINT[1,9] := MATRIX_STRUCTURE_RETAIN.MATRIX_ULINT[1,7];

    MATRIX_STRUCTURE_RETAIN.MATRIX_ULINT[2,0] := MATRIX_STRUCTURE_RETAIN.MATRIX_ULINT[2,0] + 1;
    MATRIX_STRUCTURE_RETAIN.MATRIX_ULINT[2,1] := MATRIX_STRUCTURE_RETAIN.MATRIX_ULINT[2,1] + 1;
    MATRIX_STRUCTURE_RETAIN.MATRIX_ULINT[2,2] := MATRIX_STRUCTURE_RETAIN.MATRIX_ULINT[2,2] + 1;
    MATRIX_STRUCTURE_RETAIN.MATRIX_ULINT[2,3] := MATRIX_STRUCTURE_RETAIN.MATRIX_ULINT[2,3] + 1;
    MATRIX_STRUCTURE_RETAIN.MATRIX_ULINT[2,4] := MATRIX_STRUCTURE_RETAIN.MATRIX_ULINT[2,4] + 1;
    MATRIX_STRUCTURE_RETAIN.MATRIX_ULINT[2,5] := MATRIX_STRUCTURE_RETAIN.MATRIX_ULINT[2,5] + 1;
    MATRIX_STRUCTURE_RETAIN.MATRIX_ULINT[2,6] := MATRIX_STRUCTURE_RETAIN.MATRIX_ULINT[2,6] + 1;
    MATRIX_STRUCTURE_RETAIN.MATRIX_ULINT[2,7] := MATRIX_STRUCTURE_RETAIN.MATRIX_ULINT[2,7] + 1;
    MATRIX_STRUCTURE_RETAIN.MATRIX_ULINT[2,8] := MATRIX_STRUCTURE_RETAIN.MATRIX_ULINT[2,8] + 1;
    MATRIX_STRUCTURE_RETAIN.MATRIX_ULINT[2,9] := MATRIX_STRUCTURE_RETAIN.MATRIX_ULINT[2,9] + 1;

    MATRIX_STRUCTURE_RETAIN.MATRIX_ULINT[3,0] := MATRIX_STRUCTURE_RETAIN.MATRIX_ULINT[3,0] + 1;
    MATRIX_STRUCTURE_RETAIN.MATRIX_ULINT[3,1] := MATRIX_STRUCTURE_RETAIN.MATRIX_ULINT[3,1] + 1;
    MATRIX_STRUCTURE_RETAIN.MATRIX_ULINT[3,2] := MATRIX_STRUCTURE_RETAIN.MATRIX_ULINT[3,2] + 1;
    MATRIX_STRUCTURE_RETAIN.MATRIX_ULINT[3,3] := MATRIX_STRUCTURE_RETAIN.MATRIX_ULINT[3,3] + 1;
    MATRIX_STRUCTURE_RETAIN.MATRIX_ULINT[3,4] := MATRIX_STRUCTURE_RETAIN.MATRIX_ULINT[3,4] + 1;
    MATRIX_STRUCTURE_RETAIN.MATRIX_ULINT[3,5] := MATRIX_STRUCTURE_RETAIN.MATRIX_ULINT[3,5] + 1;
    MATRIX_STRUCTURE_RETAIN.MATRIX_ULINT[3,6] := MATRIX_STRUCTURE_RETAIN.MATRIX_ULINT[3,6] + 1;
    MATRIX_STRUCTURE_RETAIN.MATRIX_ULINT[3,7] := MATRIX_STRUCTURE_RETAIN.MATRIX_ULINT[3,7] + 1;
    MATRIX_STRUCTURE_RETAIN.MATRIX_ULINT[3,8] := MATRIX_STRUCTURE_RETAIN.MATRIX_ULINT[3,8] + 1;
    MATRIX_STRUCTURE_RETAIN.MATRIX_ULINT[3,9] := MATRIX_STRUCTURE_RETAIN.MATRIX_ULINT[3,8] + 1;

    MATRIX_STRUCTURE_RETAIN.MATRIX_ULINT[4,0] := MATRIX_STRUCTURE_RETAIN.MATRIX_ULINT[4,0] + 1;
    MATRIX_STRUCTURE_RETAIN.MATRIX_ULINT[4,1] := MATRIX_STRUCTURE_RETAIN.MATRIX_ULINT[4,1] + 1;
    MATRIX_STRUCTURE_RETAIN.MATRIX_ULINT[4,2] := MATRIX_STRUCTURE_RETAIN.MATRIX_ULINT[4,2] + 1;
    MATRIX_STRUCTURE_RETAIN.MATRIX_ULINT[4,3] := MATRIX_STRUCTURE_RETAIN.MATRIX_ULINT[4,3] + 1;
    MATRIX_STRUCTURE_RETAIN.MATRIX_ULINT[4,4] := MATRIX_STRUCTURE_RETAIN.MATRIX_ULINT[4,4] + 1;
    MATRIX_STRUCTURE_RETAIN.MATRIX_ULINT[4,5] := MATRIX_STRUCTURE_RETAIN.MATRIX_ULINT[4,5] + 1;
    MATRIX_STRUCTURE_RETAIN.MATRIX_ULINT[4,6] := MATRIX_STRUCTURE_RETAIN.MATRIX_ULINT[4,6] + 1;
    MATRIX_STRUCTURE_RETAIN.MATRIX_ULINT[4,7] := MATRIX_STRUCTURE_RETAIN.MATRIX_ULINT[4,7] + 1;
    MATRIX_STRUCTURE_RETAIN.MATRIX_ULINT[4,8] := MATRIX_STRUCTURE_RETAIN.MATRIX_ULINT[4,8] + 1;
    MATRIX_STRUCTURE_RETAIN.MATRIX_ULINT[4,9] := MATRIX_STRUCTURE_RETAIN.MATRIX_ULINT[4,9] + 1;

    MATRIX_STRUCTURE_RETAIN.MATRIX_ULINT[5,0] := MATRIX_STRUCTURE_RETAIN.MATRIX_ULINT[5,0] + 1;
    MATRIX_STRUCTURE_RETAIN.MATRIX_ULINT[5,1] := MATRIX_STRUCTURE_RETAIN.MATRIX_ULINT[5,1] + 1;
    MATRIX_STRUCTURE_RETAIN.MATRIX_ULINT[5,2] := MATRIX_STRUCTURE_RETAIN.MATRIX_ULINT[5,2] + 1;
    MATRIX_STRUCTURE_RETAIN.MATRIX_ULINT[5,3] := MATRIX_STRUCTURE_RETAIN.MATRIX_ULINT[5,3] + 1;
    MATRIX_STRUCTURE_RETAIN.MATRIX_ULINT[5,4] := MATRIX_STRUCTURE_RETAIN.MATRIX_ULINT[5,4] + 1;
    MATRIX_STRUCTURE_RETAIN.MATRIX_ULINT[5,5] := MATRIX_STRUCTURE_RETAIN.MATRIX_ULINT[5,5] + 1;
    MATRIX_STRUCTURE_RETAIN.MATRIX_ULINT[5,6] := MATRIX_STRUCTURE_RETAIN.MATRIX_ULINT[5,6] + 1;
    MATRIX_STRUCTURE_RETAIN.MATRIX_ULINT[5,7] := MATRIX_STRUCTURE_RETAIN.MATRIX_ULINT[5,7] + 1;
    MATRIX_STRUCTURE_RETAIN.MATRIX_ULINT[5,8] := MATRIX_STRUCTURE_RETAIN.MATRIX_ULINT[5,8] + 1;
    MATRIX_STRUCTURE_RETAIN.MATRIX_ULINT[5,9] := MATRIX_STRUCTURE_RETAIN.MATRIX_ULINT[5,9] + 1;

    MATRIX_STRUCTURE_RETAIN.MATRIX_ULINT[6,0] := MATRIX_STRUCTURE_RETAIN.MATRIX_ULINT[6,0] + 1;
    MATRIX_STRUCTURE_RETAIN.MATRIX_ULINT[6,1] := MATRIX_STRUCTURE_RETAIN.MATRIX_ULINT[6,1] + 1;
    MATRIX_STRUCTURE_RETAIN.MATRIX_ULINT[6,2] := MATRIX_STRUCTURE_RETAIN.MATRIX_ULINT[6,2] + 1;
    MATRIX_STRUCTURE_RETAIN.MATRIX_ULINT[6,3] := MATRIX_STRUCTURE_RETAIN.MATRIX_ULINT[6,3] + 1;
    MATRIX_STRUCTURE_RETAIN.MATRIX_ULINT[6,4] := MATRIX_STRUCTURE_RETAIN.MATRIX_ULINT[6,4] + 1;
    MATRIX_STRUCTURE_RETAIN.MATRIX_ULINT[6,5] := MATRIX_STRUCTURE_RETAIN.MATRIX_ULINT[6,5] + 1;
    MATRIX_STRUCTURE_RETAIN.MATRIX_ULINT[6,6] := MATRIX_STRUCTURE_RETAIN.MATRIX_ULINT[6,6] + 1;
    MATRIX_STRUCTURE_RETAIN.MATRIX_ULINT[6,7] := MATRIX_STRUCTURE_RETAIN.MATRIX_ULINT[6,7] + 1;
    MATRIX_STRUCTURE_RETAIN.MATRIX_ULINT[6,8] := MATRIX_STRUCTURE_RETAIN.MATRIX_ULINT[6,8] + 1;
    MATRIX_STRUCTURE_RETAIN.MATRIX_ULINT[6,9] := MATRIX_STRUCTURE_RETAIN.MATRIX_ULINT[6,9] + 1;

    MATRIX_STRUCTURE_RETAIN.MATRIX_ULINT[7,0] := MATRIX_STRUCTURE_RETAIN.MATRIX_ULINT[6,0];
    MATRIX_STRUCTURE_RETAIN.MATRIX_ULINT[7,1] := MATRIX_STRUCTURE_RETAIN.MATRIX_ULINT[6,1];
    MATRIX_STRUCTURE_RETAIN.MATRIX_ULINT[7,2] := MATRIX_STRUCTURE_RETAIN.MATRIX_ULINT[6,2];
    MATRIX_STRUCTURE_RETAIN.MATRIX_ULINT[7,3] := MATRIX_STRUCTURE_RETAIN.MATRIX_ULINT[6,3];
    MATRIX_STRUCTURE_RETAIN.MATRIX_ULINT[7,4] := MATRIX_STRUCTURE_RETAIN.MATRIX_ULINT[6,4];
    MATRIX_STRUCTURE_RETAIN.MATRIX_ULINT[7,5] := MATRIX_STRUCTURE_RETAIN.MATRIX_ULINT[6,5];
    MATRIX_STRUCTURE_RETAIN.MATRIX_ULINT[7,6] := MATRIX_STRUCTURE_RETAIN.MATRIX_ULINT[6,6];
    MATRIX_STRUCTURE_RETAIN.MATRIX_ULINT[7,7] := MATRIX_STRUCTURE_RETAIN.MATRIX_ULINT[6,7];
    MATRIX_STRUCTURE_RETAIN.MATRIX_ULINT[7,8] := MATRIX_STRUCTURE_RETAIN.MATRIX_ULINT[6,8];
    MATRIX_STRUCTURE_RETAIN.MATRIX_ULINT[7,9] := MATRIX_STRUCTURE_RETAIN.MATRIX_ULINT[6,9];

    MATRIX_STRUCTURE_RETAIN.MATRIX_USINT[0,0] := MATRIX_STRUCTURE_RETAIN.MATRIX_USINT[0,0] + 1;
    MATRIX_STRUCTURE_RETAIN.MATRIX_USINT[0,1] := MATRIX_STRUCTURE_RETAIN.MATRIX_USINT[0,1] + 1;
    MATRIX_STRUCTURE_RETAIN.MATRIX_USINT[0,2] := MATRIX_STRUCTURE_RETAIN.MATRIX_USINT[0,2] + 1;
    MATRIX_STRUCTURE_RETAIN.MATRIX_USINT[0,3] := MATRIX_STRUCTURE_RETAIN.MATRIX_USINT[0,3] + 1;
    MATRIX_STRUCTURE_RETAIN.MATRIX_USINT[0,4] := MATRIX_STRUCTURE_RETAIN.MATRIX_USINT[0,4] + 1;
    MATRIX_STRUCTURE_RETAIN.MATRIX_USINT[0,5] := MATRIX_STRUCTURE_RETAIN.MATRIX_USINT[0,5] + 1;
    MATRIX_STRUCTURE_RETAIN.MATRIX_USINT[0,6] := MATRIX_STRUCTURE_RETAIN.MATRIX_USINT[0,6] + 1;
    MATRIX_STRUCTURE_RETAIN.MATRIX_USINT[0,7] := MATRIX_STRUCTURE_RETAIN.MATRIX_USINT[0,7] + 1;
    MATRIX_STRUCTURE_RETAIN.MATRIX_USINT[0,8] := MATRIX_STRUCTURE_RETAIN.MATRIX_USINT[0,6];
    MATRIX_STRUCTURE_RETAIN.MATRIX_USINT[0,9] := MATRIX_STRUCTURE_RETAIN.MATRIX_USINT[0,7];

    MATRIX_STRUCTURE_RETAIN.MATRIX_USINT[1,0] := MATRIX_STRUCTURE_RETAIN.MATRIX_USINT[1,0] + 1;
    MATRIX_STRUCTURE_RETAIN.MATRIX_USINT[1,1] := MATRIX_STRUCTURE_RETAIN.MATRIX_USINT[1,1] + 1;
    MATRIX_STRUCTURE_RETAIN.MATRIX_USINT[1,2] := MATRIX_STRUCTURE_RETAIN.MATRIX_USINT[1,2] + 1;
    MATRIX_STRUCTURE_RETAIN.MATRIX_USINT[1,3] := MATRIX_STRUCTURE_RETAIN.MATRIX_USINT[1,3] + 1;
    MATRIX_STRUCTURE_RETAIN.MATRIX_USINT[1,4] := MATRIX_STRUCTURE_RETAIN.MATRIX_USINT[1,4] + 1;
    MATRIX_STRUCTURE_RETAIN.MATRIX_USINT[1,5] := MATRIX_STRUCTURE_RETAIN.MATRIX_USINT[1,5] + 1;
    MATRIX_STRUCTURE_RETAIN.MATRIX_USINT[1,6] := MATRIX_STRUCTURE_RETAIN.MATRIX_USINT[1,6] + 1;
    MATRIX_STRUCTURE_RETAIN.MATRIX_USINT[1,7] := MATRIX_STRUCTURE_RETAIN.MATRIX_USINT[1,7] + 1;
    MATRIX_STRUCTURE_RETAIN.MATRIX_USINT[1,8] := MATRIX_STRUCTURE_RETAIN.MATRIX_USINT[1,6];
    MATRIX_STRUCTURE_RETAIN.MATRIX_USINT[1,9] := MATRIX_STRUCTURE_RETAIN.MATRIX_USINT[1,7];

    MATRIX_STRUCTURE_RETAIN.MATRIX_USINT[2,0] := MATRIX_STRUCTURE_RETAIN.MATRIX_USINT[2,0] + 1;
    MATRIX_STRUCTURE_RETAIN.MATRIX_USINT[2,1] := MATRIX_STRUCTURE_RETAIN.MATRIX_USINT[2,1] + 1;
    MATRIX_STRUCTURE_RETAIN.MATRIX_USINT[2,2] := MATRIX_STRUCTURE_RETAIN.MATRIX_USINT[2,2] + 1;
    MATRIX_STRUCTURE_RETAIN.MATRIX_USINT[2,3] := MATRIX_STRUCTURE_RETAIN.MATRIX_USINT[2,3] + 1;
    MATRIX_STRUCTURE_RETAIN.MATRIX_USINT[2,4] := MATRIX_STRUCTURE_RETAIN.MATRIX_USINT[2,4] + 1;
    MATRIX_STRUCTURE_RETAIN.MATRIX_USINT[2,5] := MATRIX_STRUCTURE_RETAIN.MATRIX_USINT[2,5] + 1;
    MATRIX_STRUCTURE_RETAIN.MATRIX_USINT[2,6] := MATRIX_STRUCTURE_RETAIN.MATRIX_USINT[2,6] + 1;
    MATRIX_STRUCTURE_RETAIN.MATRIX_USINT[2,7] := MATRIX_STRUCTURE_RETAIN.MATRIX_USINT[2,7] + 1;
    MATRIX_STRUCTURE_RETAIN.MATRIX_USINT[2,8] := MATRIX_STRUCTURE_RETAIN.MATRIX_USINT[2,8] + 1;
    MATRIX_STRUCTURE_RETAIN.MATRIX_USINT[2,9] := MATRIX_STRUCTURE_RETAIN.MATRIX_USINT[2,9] + 1;

    MATRIX_STRUCTURE_RETAIN.MATRIX_USINT[3,0] := MATRIX_STRUCTURE_RETAIN.MATRIX_USINT[3,0] + 1;
    MATRIX_STRUCTURE_RETAIN.MATRIX_USINT[3,1] := MATRIX_STRUCTURE_RETAIN.MATRIX_USINT[3,1] + 1;
    MATRIX_STRUCTURE_RETAIN.MATRIX_USINT[3,2] := MATRIX_STRUCTURE_RETAIN.MATRIX_USINT[3,2] + 1;
    MATRIX_STRUCTURE_RETAIN.MATRIX_USINT[3,3] := MATRIX_STRUCTURE_RETAIN.MATRIX_USINT[3,3] + 1;
    MATRIX_STRUCTURE_RETAIN.MATRIX_USINT[3,4] := MATRIX_STRUCTURE_RETAIN.MATRIX_USINT[3,4] + 1;
    MATRIX_STRUCTURE_RETAIN.MATRIX_USINT[3,5] := MATRIX_STRUCTURE_RETAIN.MATRIX_USINT[3,5] + 1;
    MATRIX_STRUCTURE_RETAIN.MATRIX_USINT[3,6] := MATRIX_STRUCTURE_RETAIN.MATRIX_USINT[3,6] + 1;
    MATRIX_STRUCTURE_RETAIN.MATRIX_USINT[3,7] := MATRIX_STRUCTURE_RETAIN.MATRIX_USINT[3,7] + 1;
    MATRIX_STRUCTURE_RETAIN.MATRIX_USINT[3,8] := MATRIX_STRUCTURE_RETAIN.MATRIX_USINT[3,8] + 1;
    MATRIX_STRUCTURE_RETAIN.MATRIX_USINT[3,9] := MATRIX_STRUCTURE_RETAIN.MATRIX_USINT[3,8] + 1;

    MATRIX_STRUCTURE_RETAIN.MATRIX_USINT[4,0] := MATRIX_STRUCTURE_RETAIN.MATRIX_USINT[4,0] + 1;
    MATRIX_STRUCTURE_RETAIN.MATRIX_USINT[4,1] := MATRIX_STRUCTURE_RETAIN.MATRIX_USINT[4,1] + 1;
    MATRIX_STRUCTURE_RETAIN.MATRIX_USINT[4,2] := MATRIX_STRUCTURE_RETAIN.MATRIX_USINT[4,2] + 1;
    MATRIX_STRUCTURE_RETAIN.MATRIX_USINT[4,3] := MATRIX_STRUCTURE_RETAIN.MATRIX_USINT[4,3] + 1;
    MATRIX_STRUCTURE_RETAIN.MATRIX_USINT[4,4] := MATRIX_STRUCTURE_RETAIN.MATRIX_USINT[4,4] + 1;
    MATRIX_STRUCTURE_RETAIN.MATRIX_USINT[4,5] := MATRIX_STRUCTURE_RETAIN.MATRIX_USINT[4,5] + 1;
    MATRIX_STRUCTURE_RETAIN.MATRIX_USINT[4,6] := MATRIX_STRUCTURE_RETAIN.MATRIX_USINT[4,6] + 1;
    MATRIX_STRUCTURE_RETAIN.MATRIX_USINT[4,7] := MATRIX_STRUCTURE_RETAIN.MATRIX_USINT[4,7] + 1;
    MATRIX_STRUCTURE_RETAIN.MATRIX_USINT[4,8] := MATRIX_STRUCTURE_RETAIN.MATRIX_USINT[4,8] + 1;
    MATRIX_STRUCTURE_RETAIN.MATRIX_USINT[4,9] := MATRIX_STRUCTURE_RETAIN.MATRIX_USINT[4,9] + 1;

    MATRIX_STRUCTURE_RETAIN.MATRIX_USINT[5,0] := MATRIX_STRUCTURE_RETAIN.MATRIX_USINT[5,0] + 1;
    MATRIX_STRUCTURE_RETAIN.MATRIX_USINT[5,1] := MATRIX_STRUCTURE_RETAIN.MATRIX_USINT[5,1] + 1;
    MATRIX_STRUCTURE_RETAIN.MATRIX_USINT[5,2] := MATRIX_STRUCTURE_RETAIN.MATRIX_USINT[5,2] + 1;
    MATRIX_STRUCTURE_RETAIN.MATRIX_USINT[5,3] := MATRIX_STRUCTURE_RETAIN.MATRIX_USINT[5,3] + 1;
    MATRIX_STRUCTURE_RETAIN.MATRIX_USINT[5,4] := MATRIX_STRUCTURE_RETAIN.MATRIX_USINT[5,4] + 1;
    MATRIX_STRUCTURE_RETAIN.MATRIX_USINT[5,5] := MATRIX_STRUCTURE_RETAIN.MATRIX_USINT[5,5] + 1;
    MATRIX_STRUCTURE_RETAIN.MATRIX_USINT[5,6] := MATRIX_STRUCTURE_RETAIN.MATRIX_USINT[5,6] + 1;
    MATRIX_STRUCTURE_RETAIN.MATRIX_USINT[5,7] := MATRIX_STRUCTURE_RETAIN.MATRIX_USINT[5,7] + 1;
    MATRIX_STRUCTURE_RETAIN.MATRIX_USINT[5,8] := MATRIX_STRUCTURE_RETAIN.MATRIX_USINT[5,8] + 1;
    MATRIX_STRUCTURE_RETAIN.MATRIX_USINT[5,9] := MATRIX_STRUCTURE_RETAIN.MATRIX_USINT[5,9] + 1;

    MATRIX_STRUCTURE_RETAIN.MATRIX_USINT[6,0] := MATRIX_STRUCTURE_RETAIN.MATRIX_USINT[6,0] + 1;
    MATRIX_STRUCTURE_RETAIN.MATRIX_USINT[6,1] := MATRIX_STRUCTURE_RETAIN.MATRIX_USINT[6,1] + 1;
    MATRIX_STRUCTURE_RETAIN.MATRIX_USINT[6,2] := MATRIX_STRUCTURE_RETAIN.MATRIX_USINT[6,2] + 1;
    MATRIX_STRUCTURE_RETAIN.MATRIX_USINT[6,3] := MATRIX_STRUCTURE_RETAIN.MATRIX_USINT[6,3] + 1;
    MATRIX_STRUCTURE_RETAIN.MATRIX_USINT[6,4] := MATRIX_STRUCTURE_RETAIN.MATRIX_USINT[6,4] + 1;
    MATRIX_STRUCTURE_RETAIN.MATRIX_USINT[6,5] := MATRIX_STRUCTURE_RETAIN.MATRIX_USINT[6,5] + 1;
    MATRIX_STRUCTURE_RETAIN.MATRIX_USINT[6,6] := MATRIX_STRUCTURE_RETAIN.MATRIX_USINT[6,6] + 1;
    MATRIX_STRUCTURE_RETAIN.MATRIX_USINT[6,7] := MATRIX_STRUCTURE_RETAIN.MATRIX_USINT[6,7] + 1;
    MATRIX_STRUCTURE_RETAIN.MATRIX_USINT[6,8] := MATRIX_STRUCTURE_RETAIN.MATRIX_USINT[6,8] + 1;
    MATRIX_STRUCTURE_RETAIN.MATRIX_USINT[6,9] := MATRIX_STRUCTURE_RETAIN.MATRIX_USINT[6,9] + 1;

    MATRIX_STRUCTURE_RETAIN.MATRIX_USINT[7,0] := MATRIX_STRUCTURE_RETAIN.MATRIX_USINT[6,0];
    MATRIX_STRUCTURE_RETAIN.MATRIX_USINT[7,1] := MATRIX_STRUCTURE_RETAIN.MATRIX_USINT[6,1];
    MATRIX_STRUCTURE_RETAIN.MATRIX_USINT[7,2] := MATRIX_STRUCTURE_RETAIN.MATRIX_USINT[6,2];
    MATRIX_STRUCTURE_RETAIN.MATRIX_USINT[7,3] := MATRIX_STRUCTURE_RETAIN.MATRIX_USINT[6,3];
    MATRIX_STRUCTURE_RETAIN.MATRIX_USINT[7,4] := MATRIX_STRUCTURE_RETAIN.MATRIX_USINT[6,4];
    MATRIX_STRUCTURE_RETAIN.MATRIX_USINT[7,5] := MATRIX_STRUCTURE_RETAIN.MATRIX_USINT[6,5];
    MATRIX_STRUCTURE_RETAIN.MATRIX_USINT[7,6] := MATRIX_STRUCTURE_RETAIN.MATRIX_USINT[6,6];
    MATRIX_STRUCTURE_RETAIN.MATRIX_USINT[7,7] := MATRIX_STRUCTURE_RETAIN.MATRIX_USINT[6,7];
    MATRIX_STRUCTURE_RETAIN.MATRIX_USINT[7,8] := MATRIX_STRUCTURE_RETAIN.MATRIX_USINT[6,8];
    MATRIX_STRUCTURE_RETAIN.MATRIX_USINT[7,9] := MATRIX_STRUCTURE_RETAIN.MATRIX_USINT[6,9];

    MATRIX_STRUCTURE_RETAIN.MATRIX_WORD[0,0] := MATRIX_STRUCTURE_RETAIN.MATRIX_WORD[0,0] + 1;
    MATRIX_STRUCTURE_RETAIN.MATRIX_WORD[0,1] := MATRIX_STRUCTURE_RETAIN.MATRIX_WORD[0,1] + 1;
    MATRIX_STRUCTURE_RETAIN.MATRIX_WORD[0,2] := MATRIX_STRUCTURE_RETAIN.MATRIX_WORD[0,2] + 1;
    MATRIX_STRUCTURE_RETAIN.MATRIX_WORD[0,3] := MATRIX_STRUCTURE_RETAIN.MATRIX_WORD[0,3] + 1;
    MATRIX_STRUCTURE_RETAIN.MATRIX_WORD[0,4] := MATRIX_STRUCTURE_RETAIN.MATRIX_WORD[0,4] + 1;
    MATRIX_STRUCTURE_RETAIN.MATRIX_WORD[0,5] := MATRIX_STRUCTURE_RETAIN.MATRIX_WORD[0,5] + 1;
    MATRIX_STRUCTURE_RETAIN.MATRIX_WORD[0,6] := MATRIX_STRUCTURE_RETAIN.MATRIX_WORD[0,6] + 1;
    MATRIX_STRUCTURE_RETAIN.MATRIX_WORD[0,7] := MATRIX_STRUCTURE_RETAIN.MATRIX_WORD[0,7] + 1;
    MATRIX_STRUCTURE_RETAIN.MATRIX_WORD[0,8] := MATRIX_STRUCTURE_RETAIN.MATRIX_WORD[0,6];
    MATRIX_STRUCTURE_RETAIN.MATRIX_WORD[0,9] := MATRIX_STRUCTURE_RETAIN.MATRIX_WORD[0,7];

    MATRIX_STRUCTURE_RETAIN.MATRIX_WORD[1,0] := MATRIX_STRUCTURE_RETAIN.MATRIX_WORD[1,0] + 1;
    MATRIX_STRUCTURE_RETAIN.MATRIX_WORD[1,1] := MATRIX_STRUCTURE_RETAIN.MATRIX_WORD[1,1] + 1;
    MATRIX_STRUCTURE_RETAIN.MATRIX_WORD[1,2] := MATRIX_STRUCTURE_RETAIN.MATRIX_WORD[1,2] + 1;
    MATRIX_STRUCTURE_RETAIN.MATRIX_WORD[1,3] := MATRIX_STRUCTURE_RETAIN.MATRIX_WORD[1,3] + 1;
    MATRIX_STRUCTURE_RETAIN.MATRIX_WORD[1,4] := MATRIX_STRUCTURE_RETAIN.MATRIX_WORD[1,4] + 1;
    MATRIX_STRUCTURE_RETAIN.MATRIX_WORD[1,5] := MATRIX_STRUCTURE_RETAIN.MATRIX_WORD[1,5] + 1;
    MATRIX_STRUCTURE_RETAIN.MATRIX_WORD[1,6] := MATRIX_STRUCTURE_RETAIN.MATRIX_WORD[1,6] + 1;
    MATRIX_STRUCTURE_RETAIN.MATRIX_WORD[1,7] := MATRIX_STRUCTURE_RETAIN.MATRIX_WORD[1,7] + 1;
    MATRIX_STRUCTURE_RETAIN.MATRIX_WORD[1,8] := MATRIX_STRUCTURE_RETAIN.MATRIX_WORD[1,6];
    MATRIX_STRUCTURE_RETAIN.MATRIX_WORD[1,9] := MATRIX_STRUCTURE_RETAIN.MATRIX_WORD[1,7];

    MATRIX_STRUCTURE_RETAIN.MATRIX_WORD[2,0] := MATRIX_STRUCTURE_RETAIN.MATRIX_WORD[2,0] + 1;
    MATRIX_STRUCTURE_RETAIN.MATRIX_WORD[2,1] := MATRIX_STRUCTURE_RETAIN.MATRIX_WORD[2,1] + 1;
    MATRIX_STRUCTURE_RETAIN.MATRIX_WORD[2,2] := MATRIX_STRUCTURE_RETAIN.MATRIX_WORD[2,2] + 1;
    MATRIX_STRUCTURE_RETAIN.MATRIX_WORD[2,3] := MATRIX_STRUCTURE_RETAIN.MATRIX_WORD[2,3] + 1;
    MATRIX_STRUCTURE_RETAIN.MATRIX_WORD[2,4] := MATRIX_STRUCTURE_RETAIN.MATRIX_WORD[2,4] + 1;
    MATRIX_STRUCTURE_RETAIN.MATRIX_WORD[2,5] := MATRIX_STRUCTURE_RETAIN.MATRIX_WORD[2,5] + 1;
    MATRIX_STRUCTURE_RETAIN.MATRIX_WORD[2,6] := MATRIX_STRUCTURE_RETAIN.MATRIX_WORD[2,6] + 1;
    MATRIX_STRUCTURE_RETAIN.MATRIX_WORD[2,7] := MATRIX_STRUCTURE_RETAIN.MATRIX_WORD[2,7] + 1;
    MATRIX_STRUCTURE_RETAIN.MATRIX_WORD[2,8] := MATRIX_STRUCTURE_RETAIN.MATRIX_WORD[2,8] + 1;
    MATRIX_STRUCTURE_RETAIN.MATRIX_WORD[2,9] := MATRIX_STRUCTURE_RETAIN.MATRIX_WORD[2,9] + 1;

    MATRIX_STRUCTURE_RETAIN.MATRIX_WORD[3,0] := MATRIX_STRUCTURE_RETAIN.MATRIX_WORD[3,0] + 1;
    MATRIX_STRUCTURE_RETAIN.MATRIX_WORD[3,1] := MATRIX_STRUCTURE_RETAIN.MATRIX_WORD[3,1] + 1;
    MATRIX_STRUCTURE_RETAIN.MATRIX_WORD[3,2] := MATRIX_STRUCTURE_RETAIN.MATRIX_WORD[3,2] + 1;
    MATRIX_STRUCTURE_RETAIN.MATRIX_WORD[3,3] := MATRIX_STRUCTURE_RETAIN.MATRIX_WORD[3,3] + 1;
    MATRIX_STRUCTURE_RETAIN.MATRIX_WORD[3,4] := MATRIX_STRUCTURE_RETAIN.MATRIX_WORD[3,4] + 1;
    MATRIX_STRUCTURE_RETAIN.MATRIX_WORD[3,5] := MATRIX_STRUCTURE_RETAIN.MATRIX_WORD[3,5] + 1;
    MATRIX_STRUCTURE_RETAIN.MATRIX_WORD[3,6] := MATRIX_STRUCTURE_RETAIN.MATRIX_WORD[3,6] + 1;
    MATRIX_STRUCTURE_RETAIN.MATRIX_WORD[3,7] := MATRIX_STRUCTURE_RETAIN.MATRIX_WORD[3,7] + 1;
    MATRIX_STRUCTURE_RETAIN.MATRIX_WORD[3,8] := MATRIX_STRUCTURE_RETAIN.MATRIX_WORD[3,8] + 1;
    MATRIX_STRUCTURE_RETAIN.MATRIX_WORD[3,9] := MATRIX_STRUCTURE_RETAIN.MATRIX_WORD[3,9] + 1;

    MATRIX_STRUCTURE_RETAIN.MATRIX_WORD[4,0] := MATRIX_STRUCTURE_RETAIN.MATRIX_WORD[4,0] + 1;
    MATRIX_STRUCTURE_RETAIN.MATRIX_WORD[4,1] := MATRIX_STRUCTURE_RETAIN.MATRIX_WORD[4,1] + 1;
    MATRIX_STRUCTURE_RETAIN.MATRIX_WORD[4,2] := MATRIX_STRUCTURE_RETAIN.MATRIX_WORD[4,2] + 1;
    MATRIX_STRUCTURE_RETAIN.MATRIX_WORD[4,3] := MATRIX_STRUCTURE_RETAIN.MATRIX_WORD[4,3] + 1;
    MATRIX_STRUCTURE_RETAIN.MATRIX_WORD[4,4] := MATRIX_STRUCTURE_RETAIN.MATRIX_WORD[4,4] + 1;
    MATRIX_STRUCTURE_RETAIN.MATRIX_WORD[4,5] := MATRIX_STRUCTURE_RETAIN.MATRIX_WORD[4,5] + 1;
    MATRIX_STRUCTURE_RETAIN.MATRIX_WORD[4,6] := MATRIX_STRUCTURE_RETAIN.MATRIX_WORD[4,6] + 1;
    MATRIX_STRUCTURE_RETAIN.MATRIX_WORD[4,7] := MATRIX_STRUCTURE_RETAIN.MATRIX_WORD[4,7] + 1;
    MATRIX_STRUCTURE_RETAIN.MATRIX_WORD[4,8] := MATRIX_STRUCTURE_RETAIN.MATRIX_WORD[4,8] + 1;
    MATRIX_STRUCTURE_RETAIN.MATRIX_WORD[4,9] := MATRIX_STRUCTURE_RETAIN.MATRIX_WORD[4,9] + 1;

    MATRIX_STRUCTURE_RETAIN.MATRIX_WORD[5,0] := MATRIX_STRUCTURE_RETAIN.MATRIX_WORD[5,0] + 1;
    MATRIX_STRUCTURE_RETAIN.MATRIX_WORD[5,1] := MATRIX_STRUCTURE_RETAIN.MATRIX_WORD[5,1] + 1;
    MATRIX_STRUCTURE_RETAIN.MATRIX_WORD[5,2] := MATRIX_STRUCTURE_RETAIN.MATRIX_WORD[5,2] + 1;
    MATRIX_STRUCTURE_RETAIN.MATRIX_WORD[5,3] := MATRIX_STRUCTURE_RETAIN.MATRIX_WORD[5,3] + 1;
    MATRIX_STRUCTURE_RETAIN.MATRIX_WORD[5,4] := MATRIX_STRUCTURE_RETAIN.MATRIX_WORD[5,4] + 1;
    MATRIX_STRUCTURE_RETAIN.MATRIX_WORD[5,5] := MATRIX_STRUCTURE_RETAIN.MATRIX_WORD[5,5] + 1;
    MATRIX_STRUCTURE_RETAIN.MATRIX_WORD[5,6] := MATRIX_STRUCTURE_RETAIN.MATRIX_WORD[5,6] + 1;
    MATRIX_STRUCTURE_RETAIN.MATRIX_WORD[5,7] := MATRIX_STRUCTURE_RETAIN.MATRIX_WORD[5,7] + 1;
    MATRIX_STRUCTURE_RETAIN.MATRIX_WORD[5,8] := MATRIX_STRUCTURE_RETAIN.MATRIX_WORD[5,8] + 1;
    MATRIX_STRUCTURE_RETAIN.MATRIX_WORD[5,9] := MATRIX_STRUCTURE_RETAIN.MATRIX_WORD[5,9] + 1;

    MATRIX_STRUCTURE_RETAIN.MATRIX_WORD[6,0] := MATRIX_STRUCTURE_RETAIN.MATRIX_WORD[6,0] + 1;
    MATRIX_STRUCTURE_RETAIN.MATRIX_WORD[6,1] := MATRIX_STRUCTURE_RETAIN.MATRIX_WORD[6,1] + 1;
    MATRIX_STRUCTURE_RETAIN.MATRIX_WORD[6,2] := MATRIX_STRUCTURE_RETAIN.MATRIX_WORD[6,2] + 1;
    MATRIX_STRUCTURE_RETAIN.MATRIX_WORD[6,3] := MATRIX_STRUCTURE_RETAIN.MATRIX_WORD[6,3] + 1;
    MATRIX_STRUCTURE_RETAIN.MATRIX_WORD[6,4] := MATRIX_STRUCTURE_RETAIN.MATRIX_WORD[6,4] + 1;
    MATRIX_STRUCTURE_RETAIN.MATRIX_WORD[6,5] := MATRIX_STRUCTURE_RETAIN.MATRIX_WORD[6,5] + 1;
    MATRIX_STRUCTURE_RETAIN.MATRIX_WORD[6,6] := MATRIX_STRUCTURE_RETAIN.MATRIX_WORD[6,6] + 1;
    MATRIX_STRUCTURE_RETAIN.MATRIX_WORD[6,7] := MATRIX_STRUCTURE_RETAIN.MATRIX_WORD[6,7] + 1;
    MATRIX_STRUCTURE_RETAIN.MATRIX_WORD[6,8] := MATRIX_STRUCTURE_RETAIN.MATRIX_WORD[6,8] + 1;
    MATRIX_STRUCTURE_RETAIN.MATRIX_WORD[6,9] := MATRIX_STRUCTURE_RETAIN.MATRIX_WORD[6,9] + 1;

    MATRIX_STRUCTURE_RETAIN.MATRIX_WORD[7,0] := MATRIX_STRUCTURE_RETAIN.MATRIX_WORD[6,0];
    MATRIX_STRUCTURE_RETAIN.MATRIX_WORD[7,1] := MATRIX_STRUCTURE_RETAIN.MATRIX_WORD[6,1];
    MATRIX_STRUCTURE_RETAIN.MATRIX_WORD[7,2] := MATRIX_STRUCTURE_RETAIN.MATRIX_WORD[6,2];
    MATRIX_STRUCTURE_RETAIN.MATRIX_WORD[7,3] := MATRIX_STRUCTURE_RETAIN.MATRIX_WORD[6,3];
    MATRIX_STRUCTURE_RETAIN.MATRIX_WORD[7,4] := MATRIX_STRUCTURE_RETAIN.MATRIX_WORD[6,4];
    MATRIX_STRUCTURE_RETAIN.MATRIX_WORD[7,5] := MATRIX_STRUCTURE_RETAIN.MATRIX_WORD[6,5];
    MATRIX_STRUCTURE_RETAIN.MATRIX_WORD[7,6] := MATRIX_STRUCTURE_RETAIN.MATRIX_WORD[6,6];
    MATRIX_STRUCTURE_RETAIN.MATRIX_WORD[7,7] := MATRIX_STRUCTURE_RETAIN.MATRIX_WORD[6,7];
    MATRIX_STRUCTURE_RETAIN.MATRIX_WORD[7,8] := MATRIX_STRUCTURE_RETAIN.MATRIX_WORD[6,8];
    MATRIX_STRUCTURE_RETAIN.MATRIX_WORD[7,9] := MATRIX_STRUCTURE_RETAIN.MATRIX_WORD[6,9];

    MATRIX_STRUCTURE_NON_RETAIN.MATRIX_BOOL[0,0] := NOT MATRIX_STRUCTURE_NON_RETAIN.MATRIX_BOOL[0,0];
    MATRIX_STRUCTURE_NON_RETAIN.MATRIX_BOOL[0,1] := NOT MATRIX_STRUCTURE_NON_RETAIN.MATRIX_BOOL[0,1];
    MATRIX_STRUCTURE_NON_RETAIN.MATRIX_BOOL[0,2] := NOT MATRIX_STRUCTURE_NON_RETAIN.MATRIX_BOOL[0,2];
    MATRIX_STRUCTURE_NON_RETAIN.MATRIX_BOOL[0,3] := NOT MATRIX_STRUCTURE_NON_RETAIN.MATRIX_BOOL[0,3];
    MATRIX_STRUCTURE_NON_RETAIN.MATRIX_BOOL[0,4] := NOT MATRIX_STRUCTURE_NON_RETAIN.MATRIX_BOOL[0,4];
    MATRIX_STRUCTURE_NON_RETAIN.MATRIX_BOOL[0,5] := NOT MATRIX_STRUCTURE_NON_RETAIN.MATRIX_BOOL[0,5];
    MATRIX_STRUCTURE_NON_RETAIN.MATRIX_BOOL[0,6] := NOT MATRIX_STRUCTURE_NON_RETAIN.MATRIX_BOOL[0,6];
    MATRIX_STRUCTURE_NON_RETAIN.MATRIX_BOOL[0,7] := NOT MATRIX_STRUCTURE_NON_RETAIN.MATRIX_BOOL[0,7];
    MATRIX_STRUCTURE_NON_RETAIN.MATRIX_BOOL[0,8] := MATRIX_STRUCTURE_NON_RETAIN.MATRIX_BOOL[0,6];
    MATRIX_STRUCTURE_NON_RETAIN.MATRIX_BOOL[0,9] := MATRIX_STRUCTURE_NON_RETAIN.MATRIX_BOOL[0,7];

    MATRIX_STRUCTURE_NON_RETAIN.MATRIX_BOOL[1,0] := NOT MATRIX_STRUCTURE_NON_RETAIN.MATRIX_BOOL[1,0];
    MATRIX_STRUCTURE_NON_RETAIN.MATRIX_BOOL[1,1] := NOT MATRIX_STRUCTURE_NON_RETAIN.MATRIX_BOOL[1,1];
    MATRIX_STRUCTURE_NON_RETAIN.MATRIX_BOOL[1,2] := NOT MATRIX_STRUCTURE_NON_RETAIN.MATRIX_BOOL[1,2];
    MATRIX_STRUCTURE_NON_RETAIN.MATRIX_BOOL[1,3] := NOT MATRIX_STRUCTURE_NON_RETAIN.MATRIX_BOOL[1,3];
    MATRIX_STRUCTURE_NON_RETAIN.MATRIX_BOOL[1,4] := NOT MATRIX_STRUCTURE_NON_RETAIN.MATRIX_BOOL[1,4];
    MATRIX_STRUCTURE_NON_RETAIN.MATRIX_BOOL[1,5] := NOT MATRIX_STRUCTURE_NON_RETAIN.MATRIX_BOOL[1,5];
    MATRIX_STRUCTURE_NON_RETAIN.MATRIX_BOOL[1,6] := NOT MATRIX_STRUCTURE_NON_RETAIN.MATRIX_BOOL[1,6];
    MATRIX_STRUCTURE_NON_RETAIN.MATRIX_BOOL[1,7] := NOT MATRIX_STRUCTURE_NON_RETAIN.MATRIX_BOOL[1,7];
    MATRIX_STRUCTURE_NON_RETAIN.MATRIX_BOOL[1,8] := MATRIX_STRUCTURE_NON_RETAIN.MATRIX_BOOL[1,6];
    MATRIX_STRUCTURE_NON_RETAIN.MATRIX_BOOL[1,9] := MATRIX_STRUCTURE_NON_RETAIN.MATRIX_BOOL[1,7];

    MATRIX_STRUCTURE_NON_RETAIN.MATRIX_BOOL[2,0] := NOT MATRIX_STRUCTURE_NON_RETAIN.MATRIX_BOOL[2,0];
    MATRIX_STRUCTURE_NON_RETAIN.MATRIX_BOOL[2,1] := NOT MATRIX_STRUCTURE_NON_RETAIN.MATRIX_BOOL[2,1];
    MATRIX_STRUCTURE_NON_RETAIN.MATRIX_BOOL[2,2] := NOT MATRIX_STRUCTURE_NON_RETAIN.MATRIX_BOOL[2,2];
    MATRIX_STRUCTURE_NON_RETAIN.MATRIX_BOOL[2,3] := NOT MATRIX_STRUCTURE_NON_RETAIN.MATRIX_BOOL[2,3];
    MATRIX_STRUCTURE_NON_RETAIN.MATRIX_BOOL[2,4] := NOT MATRIX_STRUCTURE_NON_RETAIN.MATRIX_BOOL[2,4];
    MATRIX_STRUCTURE_NON_RETAIN.MATRIX_BOOL[2,5] := NOT MATRIX_STRUCTURE_NON_RETAIN.MATRIX_BOOL[2,5];
    MATRIX_STRUCTURE_NON_RETAIN.MATRIX_BOOL[2,6] := NOT MATRIX_STRUCTURE_NON_RETAIN.MATRIX_BOOL[2,6];
    MATRIX_STRUCTURE_NON_RETAIN.MATRIX_BOOL[2,7] := NOT MATRIX_STRUCTURE_NON_RETAIN.MATRIX_BOOL[2,7];
    MATRIX_STRUCTURE_NON_RETAIN.MATRIX_BOOL[2,8] := NOT MATRIX_STRUCTURE_NON_RETAIN.MATRIX_BOOL[2,8];
    MATRIX_STRUCTURE_NON_RETAIN.MATRIX_BOOL[2,9] := NOT MATRIX_STRUCTURE_NON_RETAIN.MATRIX_BOOL[2,9];

    MATRIX_STRUCTURE_NON_RETAIN.MATRIX_BOOL[3,0] := NOT MATRIX_STRUCTURE_NON_RETAIN.MATRIX_BOOL[3,0];
    MATRIX_STRUCTURE_NON_RETAIN.MATRIX_BOOL[3,1] := NOT MATRIX_STRUCTURE_NON_RETAIN.MATRIX_BOOL[3,1];
    MATRIX_STRUCTURE_NON_RETAIN.MATRIX_BOOL[3,2] := NOT MATRIX_STRUCTURE_NON_RETAIN.MATRIX_BOOL[3,2];
    MATRIX_STRUCTURE_NON_RETAIN.MATRIX_BOOL[3,3] := NOT MATRIX_STRUCTURE_NON_RETAIN.MATRIX_BOOL[3,3];
    MATRIX_STRUCTURE_NON_RETAIN.MATRIX_BOOL[3,4] := NOT MATRIX_STRUCTURE_NON_RETAIN.MATRIX_BOOL[3,4];
    MATRIX_STRUCTURE_NON_RETAIN.MATRIX_BOOL[3,5] := NOT MATRIX_STRUCTURE_NON_RETAIN.MATRIX_BOOL[3,5];
    MATRIX_STRUCTURE_NON_RETAIN.MATRIX_BOOL[3,6] := NOT MATRIX_STRUCTURE_NON_RETAIN.MATRIX_BOOL[3,6];
    MATRIX_STRUCTURE_NON_RETAIN.MATRIX_BOOL[3,7] := NOT MATRIX_STRUCTURE_NON_RETAIN.MATRIX_BOOL[3,7];
    MATRIX_STRUCTURE_NON_RETAIN.MATRIX_BOOL[3,8] := NOT MATRIX_STRUCTURE_NON_RETAIN.MATRIX_BOOL[3,8];
    MATRIX_STRUCTURE_NON_RETAIN.MATRIX_BOOL[3,9] := NOT MATRIX_STRUCTURE_NON_RETAIN.MATRIX_BOOL[3,9];

    MATRIX_STRUCTURE_NON_RETAIN.MATRIX_BOOL[4,0] := NOT MATRIX_STRUCTURE_NON_RETAIN.MATRIX_BOOL[4,0];
    MATRIX_STRUCTURE_NON_RETAIN.MATRIX_BOOL[4,1] := NOT MATRIX_STRUCTURE_NON_RETAIN.MATRIX_BOOL[4,1];
    MATRIX_STRUCTURE_NON_RETAIN.MATRIX_BOOL[4,2] := NOT MATRIX_STRUCTURE_NON_RETAIN.MATRIX_BOOL[4,2];
    MATRIX_STRUCTURE_NON_RETAIN.MATRIX_BOOL[4,3] := NOT MATRIX_STRUCTURE_NON_RETAIN.MATRIX_BOOL[4,3];
    MATRIX_STRUCTURE_NON_RETAIN.MATRIX_BOOL[4,4] := NOT MATRIX_STRUCTURE_NON_RETAIN.MATRIX_BOOL[4,4];
    MATRIX_STRUCTURE_NON_RETAIN.MATRIX_BOOL[4,5] := NOT MATRIX_STRUCTURE_NON_RETAIN.MATRIX_BOOL[4,5];
    MATRIX_STRUCTURE_NON_RETAIN.MATRIX_BOOL[4,6] := NOT MATRIX_STRUCTURE_NON_RETAIN.MATRIX_BOOL[4,6];
    MATRIX_STRUCTURE_NON_RETAIN.MATRIX_BOOL[4,7] := NOT MATRIX_STRUCTURE_NON_RETAIN.MATRIX_BOOL[4,7];
    MATRIX_STRUCTURE_NON_RETAIN.MATRIX_BOOL[4,8] := NOT MATRIX_STRUCTURE_NON_RETAIN.MATRIX_BOOL[4,8];
    MATRIX_STRUCTURE_NON_RETAIN.MATRIX_BOOL[4,9] := NOT MATRIX_STRUCTURE_NON_RETAIN.MATRIX_BOOL[4,9];

    MATRIX_STRUCTURE_NON_RETAIN.MATRIX_BOOL[5,0] := NOT MATRIX_STRUCTURE_NON_RETAIN.MATRIX_BOOL[5,0];
    MATRIX_STRUCTURE_NON_RETAIN.MATRIX_BOOL[5,1] := NOT MATRIX_STRUCTURE_NON_RETAIN.MATRIX_BOOL[5,1];
    MATRIX_STRUCTURE_NON_RETAIN.MATRIX_BOOL[5,2] := NOT MATRIX_STRUCTURE_NON_RETAIN.MATRIX_BOOL[5,2];
    MATRIX_STRUCTURE_NON_RETAIN.MATRIX_BOOL[5,3] := NOT MATRIX_STRUCTURE_NON_RETAIN.MATRIX_BOOL[5,3];
    MATRIX_STRUCTURE_NON_RETAIN.MATRIX_BOOL[5,4] := NOT MATRIX_STRUCTURE_NON_RETAIN.MATRIX_BOOL[5,4];
    MATRIX_STRUCTURE_NON_RETAIN.MATRIX_BOOL[5,5] := NOT MATRIX_STRUCTURE_NON_RETAIN.MATRIX_BOOL[5,5];
    MATRIX_STRUCTURE_NON_RETAIN.MATRIX_BOOL[5,6] := NOT MATRIX_STRUCTURE_NON_RETAIN.MATRIX_BOOL[5,6];
    MATRIX_STRUCTURE_NON_RETAIN.MATRIX_BOOL[5,7] := NOT MATRIX_STRUCTURE_NON_RETAIN.MATRIX_BOOL[5,7];
    MATRIX_STRUCTURE_NON_RETAIN.MATRIX_BOOL[5,8] := NOT MATRIX_STRUCTURE_NON_RETAIN.MATRIX_BOOL[5,8];
    MATRIX_STRUCTURE_NON_RETAIN.MATRIX_BOOL[5,9] := NOT MATRIX_STRUCTURE_NON_RETAIN.MATRIX_BOOL[5,9];

    MATRIX_STRUCTURE_NON_RETAIN.MATRIX_BOOL[6,0] := NOT MATRIX_STRUCTURE_NON_RETAIN.MATRIX_BOOL[6,0];
    MATRIX_STRUCTURE_NON_RETAIN.MATRIX_BOOL[6,1] := NOT MATRIX_STRUCTURE_NON_RETAIN.MATRIX_BOOL[6,1];
    MATRIX_STRUCTURE_NON_RETAIN.MATRIX_BOOL[6,2] := NOT MATRIX_STRUCTURE_NON_RETAIN.MATRIX_BOOL[6,2];
    MATRIX_STRUCTURE_NON_RETAIN.MATRIX_BOOL[6,3] := NOT MATRIX_STRUCTURE_NON_RETAIN.MATRIX_BOOL[6,3];
    MATRIX_STRUCTURE_NON_RETAIN.MATRIX_BOOL[6,4] := NOT MATRIX_STRUCTURE_NON_RETAIN.MATRIX_BOOL[6,4];
    MATRIX_STRUCTURE_NON_RETAIN.MATRIX_BOOL[6,5] := NOT MATRIX_STRUCTURE_NON_RETAIN.MATRIX_BOOL[6,5];
    MATRIX_STRUCTURE_NON_RETAIN.MATRIX_BOOL[6,6] := NOT MATRIX_STRUCTURE_NON_RETAIN.MATRIX_BOOL[6,6];
    MATRIX_STRUCTURE_NON_RETAIN.MATRIX_BOOL[6,7] := NOT MATRIX_STRUCTURE_NON_RETAIN.MATRIX_BOOL[6,7];
    MATRIX_STRUCTURE_NON_RETAIN.MATRIX_BOOL[6,8] := NOT MATRIX_STRUCTURE_NON_RETAIN.MATRIX_BOOL[6,8];
    MATRIX_STRUCTURE_NON_RETAIN.MATRIX_BOOL[6,9] := NOT MATRIX_STRUCTURE_NON_RETAIN.MATRIX_BOOL[6,9];

    MATRIX_STRUCTURE_NON_RETAIN.MATRIX_BOOL[7,0] := MATRIX_STRUCTURE_NON_RETAIN.MATRIX_BOOL[6,0];
    MATRIX_STRUCTURE_NON_RETAIN.MATRIX_BOOL[7,1] := MATRIX_STRUCTURE_NON_RETAIN.MATRIX_BOOL[6,1];
    MATRIX_STRUCTURE_NON_RETAIN.MATRIX_BOOL[7,2] := MATRIX_STRUCTURE_NON_RETAIN.MATRIX_BOOL[6,2];
    MATRIX_STRUCTURE_NON_RETAIN.MATRIX_BOOL[7,3] := MATRIX_STRUCTURE_NON_RETAIN.MATRIX_BOOL[6,3];
    MATRIX_STRUCTURE_NON_RETAIN.MATRIX_BOOL[7,4] := MATRIX_STRUCTURE_NON_RETAIN.MATRIX_BOOL[6,4];
    MATRIX_STRUCTURE_NON_RETAIN.MATRIX_BOOL[7,5] := MATRIX_STRUCTURE_NON_RETAIN.MATRIX_BOOL[6,5];
    MATRIX_STRUCTURE_NON_RETAIN.MATRIX_BOOL[7,6] := MATRIX_STRUCTURE_NON_RETAIN.MATRIX_BOOL[6,6];
    MATRIX_STRUCTURE_NON_RETAIN.MATRIX_BOOL[7,7] := MATRIX_STRUCTURE_NON_RETAIN.MATRIX_BOOL[6,7];
    MATRIX_STRUCTURE_NON_RETAIN.MATRIX_BOOL[7,8] := MATRIX_STRUCTURE_NON_RETAIN.MATRIX_BOOL[6,8];
    MATRIX_STRUCTURE_NON_RETAIN.MATRIX_BOOL[7,9] := MATRIX_STRUCTURE_NON_RETAIN.MATRIX_BOOL[6,9];

    MATRIX_STRUCTURE_NON_RETAIN.MATRIX_BYTE[0,0] := MATRIX_STRUCTURE_NON_RETAIN.MATRIX_BYTE[0,0] + 1;
    MATRIX_STRUCTURE_NON_RETAIN.MATRIX_BYTE[0,1] := MATRIX_STRUCTURE_NON_RETAIN.MATRIX_BYTE[0,1] + 1;
    MATRIX_STRUCTURE_NON_RETAIN.MATRIX_BYTE[0,2] := MATRIX_STRUCTURE_NON_RETAIN.MATRIX_BYTE[0,2] + 1;
    MATRIX_STRUCTURE_NON_RETAIN.MATRIX_BYTE[0,3] := MATRIX_STRUCTURE_NON_RETAIN.MATRIX_BYTE[0,3] + 1;
    MATRIX_STRUCTURE_NON_RETAIN.MATRIX_BYTE[0,4] := MATRIX_STRUCTURE_NON_RETAIN.MATRIX_BYTE[0,4] + 1;
    MATRIX_STRUCTURE_NON_RETAIN.MATRIX_BYTE[0,5] := MATRIX_STRUCTURE_NON_RETAIN.MATRIX_BYTE[0,5] + 1;
    MATRIX_STRUCTURE_NON_RETAIN.MATRIX_BYTE[0,6] := MATRIX_STRUCTURE_NON_RETAIN.MATRIX_BYTE[0,6] + 1;
    MATRIX_STRUCTURE_NON_RETAIN.MATRIX_BYTE[0,7] := MATRIX_STRUCTURE_NON_RETAIN.MATRIX_BYTE[0,7] + 1;
    MATRIX_STRUCTURE_NON_RETAIN.MATRIX_BYTE[0,8] := MATRIX_STRUCTURE_NON_RETAIN.MATRIX_BYTE[0,6];
    MATRIX_STRUCTURE_NON_RETAIN.MATRIX_BYTE[0,9] := MATRIX_STRUCTURE_NON_RETAIN.MATRIX_BYTE[0,7];

    MATRIX_STRUCTURE_NON_RETAIN.MATRIX_BYTE[1,0] := MATRIX_STRUCTURE_NON_RETAIN.MATRIX_BYTE[1,0] + 1;
    MATRIX_STRUCTURE_NON_RETAIN.MATRIX_BYTE[1,1] := MATRIX_STRUCTURE_NON_RETAIN.MATRIX_BYTE[1,1] + 1;
    MATRIX_STRUCTURE_NON_RETAIN.MATRIX_BYTE[1,2] := MATRIX_STRUCTURE_NON_RETAIN.MATRIX_BYTE[1,2] + 1;
    MATRIX_STRUCTURE_NON_RETAIN.MATRIX_BYTE[1,3] := MATRIX_STRUCTURE_NON_RETAIN.MATRIX_BYTE[1,3] + 1;
    MATRIX_STRUCTURE_NON_RETAIN.MATRIX_BYTE[1,4] := MATRIX_STRUCTURE_NON_RETAIN.MATRIX_BYTE[1,4] + 1;
    MATRIX_STRUCTURE_NON_RETAIN.MATRIX_BYTE[1,5] := MATRIX_STRUCTURE_NON_RETAIN.MATRIX_BYTE[1,5] + 1;
    MATRIX_STRUCTURE_NON_RETAIN.MATRIX_BYTE[1,6] := MATRIX_STRUCTURE_NON_RETAIN.MATRIX_BYTE[1,6] + 1;
    MATRIX_STRUCTURE_NON_RETAIN.MATRIX_BYTE[1,7] := MATRIX_STRUCTURE_NON_RETAIN.MATRIX_BYTE[1,7] + 1;
    MATRIX_STRUCTURE_NON_RETAIN.MATRIX_BYTE[1,8] := MATRIX_STRUCTURE_NON_RETAIN.MATRIX_BYTE[1,6];
    MATRIX_STRUCTURE_NON_RETAIN.MATRIX_BYTE[1,9] := MATRIX_STRUCTURE_NON_RETAIN.MATRIX_BYTE[1,7];

    MATRIX_STRUCTURE_NON_RETAIN.MATRIX_BYTE[2,0] := MATRIX_STRUCTURE_NON_RETAIN.MATRIX_BYTE[2,0] + 1;
    MATRIX_STRUCTURE_NON_RETAIN.MATRIX_BYTE[2,1] := MATRIX_STRUCTURE_NON_RETAIN.MATRIX_BYTE[2,1] + 1;
    MATRIX_STRUCTURE_NON_RETAIN.MATRIX_BYTE[2,2] := MATRIX_STRUCTURE_NON_RETAIN.MATRIX_BYTE[2,2] + 1;
    MATRIX_STRUCTURE_NON_RETAIN.MATRIX_BYTE[2,3] := MATRIX_STRUCTURE_NON_RETAIN.MATRIX_BYTE[2,3] + 1;
    MATRIX_STRUCTURE_NON_RETAIN.MATRIX_BYTE[2,4] := MATRIX_STRUCTURE_NON_RETAIN.MATRIX_BYTE[2,4] + 1;
    MATRIX_STRUCTURE_NON_RETAIN.MATRIX_BYTE[2,5] := MATRIX_STRUCTURE_NON_RETAIN.MATRIX_BYTE[2,5] + 1;
    MATRIX_STRUCTURE_NON_RETAIN.MATRIX_BYTE[2,6] := MATRIX_STRUCTURE_NON_RETAIN.MATRIX_BYTE[2,6] + 1;
    MATRIX_STRUCTURE_NON_RETAIN.MATRIX_BYTE[2,7] := MATRIX_STRUCTURE_NON_RETAIN.MATRIX_BYTE[2,7] + 1;
    MATRIX_STRUCTURE_NON_RETAIN.MATRIX_BYTE[2,8] := MATRIX_STRUCTURE_NON_RETAIN.MATRIX_BYTE[2,8] + 1;
    MATRIX_STRUCTURE_NON_RETAIN.MATRIX_BYTE[2,9] := MATRIX_STRUCTURE_NON_RETAIN.MATRIX_BYTE[2,9] + 1;

    MATRIX_STRUCTURE_NON_RETAIN.MATRIX_BYTE[3,0] := MATRIX_STRUCTURE_NON_RETAIN.MATRIX_BYTE[3,0] + 1;
    MATRIX_STRUCTURE_NON_RETAIN.MATRIX_BYTE[3,1] := MATRIX_STRUCTURE_NON_RETAIN.MATRIX_BYTE[3,1] + 1;
    MATRIX_STRUCTURE_NON_RETAIN.MATRIX_BYTE[3,2] := MATRIX_STRUCTURE_NON_RETAIN.MATRIX_BYTE[3,2] + 1;
    MATRIX_STRUCTURE_NON_RETAIN.MATRIX_BYTE[3,3] := MATRIX_STRUCTURE_NON_RETAIN.MATRIX_BYTE[3,3] + 1;
    MATRIX_STRUCTURE_NON_RETAIN.MATRIX_BYTE[3,4] := MATRIX_STRUCTURE_NON_RETAIN.MATRIX_BYTE[3,4] + 1;
    MATRIX_STRUCTURE_NON_RETAIN.MATRIX_BYTE[3,5] := MATRIX_STRUCTURE_NON_RETAIN.MATRIX_BYTE[3,5] + 1;
    MATRIX_STRUCTURE_NON_RETAIN.MATRIX_BYTE[3,6] := MATRIX_STRUCTURE_NON_RETAIN.MATRIX_BYTE[3,6] + 1;
    MATRIX_STRUCTURE_NON_RETAIN.MATRIX_BYTE[3,7] := MATRIX_STRUCTURE_NON_RETAIN.MATRIX_BYTE[3,7] + 1;
    MATRIX_STRUCTURE_NON_RETAIN.MATRIX_BYTE[3,8] := MATRIX_STRUCTURE_NON_RETAIN.MATRIX_BYTE[3,8] + 1;
    MATRIX_STRUCTURE_NON_RETAIN.MATRIX_BYTE[3,9] := MATRIX_STRUCTURE_NON_RETAIN.MATRIX_BYTE[3,9] + 1;

    MATRIX_STRUCTURE_NON_RETAIN.MATRIX_BYTE[4,0] := MATRIX_STRUCTURE_NON_RETAIN.MATRIX_BYTE[4,0] + 1;
    MATRIX_STRUCTURE_NON_RETAIN.MATRIX_BYTE[4,1] := MATRIX_STRUCTURE_NON_RETAIN.MATRIX_BYTE[4,1] + 1;
    MATRIX_STRUCTURE_NON_RETAIN.MATRIX_BYTE[4,2] := MATRIX_STRUCTURE_NON_RETAIN.MATRIX_BYTE[4,2] + 1;
    MATRIX_STRUCTURE_NON_RETAIN.MATRIX_BYTE[4,3] := MATRIX_STRUCTURE_NON_RETAIN.MATRIX_BYTE[4,3] + 1;
    MATRIX_STRUCTURE_NON_RETAIN.MATRIX_BYTE[4,4] := MATRIX_STRUCTURE_NON_RETAIN.MATRIX_BYTE[4,4] + 1;
    MATRIX_STRUCTURE_NON_RETAIN.MATRIX_BYTE[4,5] := MATRIX_STRUCTURE_NON_RETAIN.MATRIX_BYTE[4,5] + 1;
    MATRIX_STRUCTURE_NON_RETAIN.MATRIX_BYTE[4,6] := MATRIX_STRUCTURE_NON_RETAIN.MATRIX_BYTE[4,6] + 1;
    MATRIX_STRUCTURE_NON_RETAIN.MATRIX_BYTE[4,7] := MATRIX_STRUCTURE_NON_RETAIN.MATRIX_BYTE[4,7] + 1;
    MATRIX_STRUCTURE_NON_RETAIN.MATRIX_BYTE[4,8] := MATRIX_STRUCTURE_NON_RETAIN.MATRIX_BYTE[4,8] + 1;
    MATRIX_STRUCTURE_NON_RETAIN.MATRIX_BYTE[4,9] := MATRIX_STRUCTURE_NON_RETAIN.MATRIX_BYTE[4,9] + 1;

    MATRIX_STRUCTURE_NON_RETAIN.MATRIX_BYTE[5,0] := MATRIX_STRUCTURE_NON_RETAIN.MATRIX_BYTE[5,0] + 1;
    MATRIX_STRUCTURE_NON_RETAIN.MATRIX_BYTE[5,1] := MATRIX_STRUCTURE_NON_RETAIN.MATRIX_BYTE[5,1] + 1;
    MATRIX_STRUCTURE_NON_RETAIN.MATRIX_BYTE[5,2] := MATRIX_STRUCTURE_NON_RETAIN.MATRIX_BYTE[5,2] + 1;
    MATRIX_STRUCTURE_NON_RETAIN.MATRIX_BYTE[5,3] := MATRIX_STRUCTURE_NON_RETAIN.MATRIX_BYTE[5,3] + 1;
    MATRIX_STRUCTURE_NON_RETAIN.MATRIX_BYTE[5,4] := MATRIX_STRUCTURE_NON_RETAIN.MATRIX_BYTE[5,4] + 1;
    MATRIX_STRUCTURE_NON_RETAIN.MATRIX_BYTE[5,5] := MATRIX_STRUCTURE_NON_RETAIN.MATRIX_BYTE[5,5] + 1;
    MATRIX_STRUCTURE_NON_RETAIN.MATRIX_BYTE[5,6] := MATRIX_STRUCTURE_NON_RETAIN.MATRIX_BYTE[5,6] + 1;
    MATRIX_STRUCTURE_NON_RETAIN.MATRIX_BYTE[5,7] := MATRIX_STRUCTURE_NON_RETAIN.MATRIX_BYTE[5,7] + 1;
    MATRIX_STRUCTURE_NON_RETAIN.MATRIX_BYTE[5,8] := MATRIX_STRUCTURE_NON_RETAIN.MATRIX_BYTE[5,8] + 1;
    MATRIX_STRUCTURE_NON_RETAIN.MATRIX_BYTE[5,9] := MATRIX_STRUCTURE_NON_RETAIN.MATRIX_BYTE[5,9] + 1;

    MATRIX_STRUCTURE_NON_RETAIN.MATRIX_BYTE[6,0] := MATRIX_STRUCTURE_NON_RETAIN.MATRIX_BYTE[6,0] + 1;
    MATRIX_STRUCTURE_NON_RETAIN.MATRIX_BYTE[6,1] := MATRIX_STRUCTURE_NON_RETAIN.MATRIX_BYTE[6,1] + 1;
    MATRIX_STRUCTURE_NON_RETAIN.MATRIX_BYTE[6,2] := MATRIX_STRUCTURE_NON_RETAIN.MATRIX_BYTE[6,2] + 1;
    MATRIX_STRUCTURE_NON_RETAIN.MATRIX_BYTE[6,3] := MATRIX_STRUCTURE_NON_RETAIN.MATRIX_BYTE[6,3] + 1;
    MATRIX_STRUCTURE_NON_RETAIN.MATRIX_BYTE[6,4] := MATRIX_STRUCTURE_NON_RETAIN.MATRIX_BYTE[6,4] + 1;
    MATRIX_STRUCTURE_NON_RETAIN.MATRIX_BYTE[6,5] := MATRIX_STRUCTURE_NON_RETAIN.MATRIX_BYTE[6,5] + 1;
    MATRIX_STRUCTURE_NON_RETAIN.MATRIX_BYTE[6,6] := MATRIX_STRUCTURE_NON_RETAIN.MATRIX_BYTE[6,6] + 1;
    MATRIX_STRUCTURE_NON_RETAIN.MATRIX_BYTE[6,7] := MATRIX_STRUCTURE_NON_RETAIN.MATRIX_BYTE[6,7] + 1;
    MATRIX_STRUCTURE_NON_RETAIN.MATRIX_BYTE[6,8] := MATRIX_STRUCTURE_NON_RETAIN.MATRIX_BYTE[6,8] + 1;
    MATRIX_STRUCTURE_NON_RETAIN.MATRIX_BYTE[6,9] := MATRIX_STRUCTURE_NON_RETAIN.MATRIX_BYTE[6,9] + 1;

    MATRIX_STRUCTURE_NON_RETAIN.MATRIX_BYTE[7,0] := MATRIX_STRUCTURE_NON_RETAIN.MATRIX_BYTE[6,0];
    MATRIX_STRUCTURE_NON_RETAIN.MATRIX_BYTE[7,1] := MATRIX_STRUCTURE_NON_RETAIN.MATRIX_BYTE[6,1];
    MATRIX_STRUCTURE_NON_RETAIN.MATRIX_BYTE[7,2] := MATRIX_STRUCTURE_NON_RETAIN.MATRIX_BYTE[6,2];
    MATRIX_STRUCTURE_NON_RETAIN.MATRIX_BYTE[7,3] := MATRIX_STRUCTURE_NON_RETAIN.MATRIX_BYTE[6,3];
    MATRIX_STRUCTURE_NON_RETAIN.MATRIX_BYTE[7,4] := MATRIX_STRUCTURE_NON_RETAIN.MATRIX_BYTE[6,4];
    MATRIX_STRUCTURE_NON_RETAIN.MATRIX_BYTE[7,5] := MATRIX_STRUCTURE_NON_RETAIN.MATRIX_BYTE[6,5];
    MATRIX_STRUCTURE_NON_RETAIN.MATRIX_BYTE[7,6] := MATRIX_STRUCTURE_NON_RETAIN.MATRIX_BYTE[6,6];
    MATRIX_STRUCTURE_NON_RETAIN.MATRIX_BYTE[7,7] := MATRIX_STRUCTURE_NON_RETAIN.MATRIX_BYTE[6,7];
    MATRIX_STRUCTURE_NON_RETAIN.MATRIX_BYTE[7,8] := MATRIX_STRUCTURE_NON_RETAIN.MATRIX_BYTE[6,8];
    MATRIX_STRUCTURE_NON_RETAIN.MATRIX_BYTE[7,9] := MATRIX_STRUCTURE_NON_RETAIN.MATRIX_BYTE[6,9];

    MATRIX_STRUCTURE_NON_RETAIN.MATRIX_DATE[0,0] := ANY_TO_DATE(1445385600 + MATRIX_STRUCTURE_NON_RETAIN.MATRIX_DINT[0,0] * 86400);
    MATRIX_STRUCTURE_NON_RETAIN.MATRIX_DATE[0,1] := ANY_TO_DATE(1445385600 + MATRIX_STRUCTURE_NON_RETAIN.MATRIX_DINT[0,1] * 86400);
    MATRIX_STRUCTURE_NON_RETAIN.MATRIX_DATE[0,2] := ANY_TO_DATE(1445385600 + MATRIX_STRUCTURE_NON_RETAIN.MATRIX_DINT[0,2] * 86400);
    MATRIX_STRUCTURE_NON_RETAIN.MATRIX_DATE[0,3] := ANY_TO_DATE(1445385600 + MATRIX_STRUCTURE_NON_RETAIN.MATRIX_DINT[0,3] * 86400);
    MATRIX_STRUCTURE_NON_RETAIN.MATRIX_DATE[0,4] := ANY_TO_DATE(1445385600 + MATRIX_STRUCTURE_NON_RETAIN.MATRIX_DINT[0,4] * 86400);
    MATRIX_STRUCTURE_NON_RETAIN.MATRIX_DATE[0,5] := ANY_TO_DATE(1445385600 + MATRIX_STRUCTURE_NON_RETAIN.MATRIX_DINT[0,5] * 86400);
    MATRIX_STRUCTURE_NON_RETAIN.MATRIX_DATE[0,6] := ANY_TO_DATE(1445385600 + MATRIX_STRUCTURE_NON_RETAIN.MATRIX_DINT[0,6] * 86400);
    MATRIX_STRUCTURE_NON_RETAIN.MATRIX_DATE[0,7] := ANY_TO_DATE(1445385600 + MATRIX_STRUCTURE_NON_RETAIN.MATRIX_DINT[0,7] * 86400);
    MATRIX_STRUCTURE_NON_RETAIN.MATRIX_DATE[0,8] := MATRIX_STRUCTURE_NON_RETAIN.MATRIX_DATE[0,6];
    MATRIX_STRUCTURE_NON_RETAIN.MATRIX_DATE[0,9] := MATRIX_STRUCTURE_NON_RETAIN.MATRIX_DATE[0,7];

    MATRIX_STRUCTURE_NON_RETAIN.MATRIX_DATE[1,0] := ANY_TO_DATE(1445385600 + MATRIX_STRUCTURE_NON_RETAIN.MATRIX_DINT[1,0] * 86400);
    MATRIX_STRUCTURE_NON_RETAIN.MATRIX_DATE[1,1] := ANY_TO_DATE(1445385600 + MATRIX_STRUCTURE_NON_RETAIN.MATRIX_DINT[1,1] * 86400);
    MATRIX_STRUCTURE_NON_RETAIN.MATRIX_DATE[1,2] := ANY_TO_DATE(1445385600 + MATRIX_STRUCTURE_NON_RETAIN.MATRIX_DINT[1,2] * 86400);
    MATRIX_STRUCTURE_NON_RETAIN.MATRIX_DATE[1,3] := ANY_TO_DATE(1445385600 + MATRIX_STRUCTURE_NON_RETAIN.MATRIX_DINT[1,3] * 86400);
    MATRIX_STRUCTURE_NON_RETAIN.MATRIX_DATE[1,4] := ANY_TO_DATE(1445385600 + MATRIX_STRUCTURE_NON_RETAIN.MATRIX_DINT[1,4] * 86400);
    MATRIX_STRUCTURE_NON_RETAIN.MATRIX_DATE[1,5] := ANY_TO_DATE(1445385600 + MATRIX_STRUCTURE_NON_RETAIN.MATRIX_DINT[1,5] * 86400);
    MATRIX_STRUCTURE_NON_RETAIN.MATRIX_DATE[1,6] := ANY_TO_DATE(1445385600 + MATRIX_STRUCTURE_NON_RETAIN.MATRIX_DINT[1,6] * 86400);
    MATRIX_STRUCTURE_NON_RETAIN.MATRIX_DATE[1,7] := ANY_TO_DATE(1445385600 + MATRIX_STRUCTURE_NON_RETAIN.MATRIX_DINT[1,7] * 86400);
    MATRIX_STRUCTURE_NON_RETAIN.MATRIX_DATE[1,8] := MATRIX_STRUCTURE_NON_RETAIN.MATRIX_DATE[1,6];
    MATRIX_STRUCTURE_NON_RETAIN.MATRIX_DATE[1,9] := MATRIX_STRUCTURE_NON_RETAIN.MATRIX_DATE[1,7];

    MATRIX_STRUCTURE_NON_RETAIN.MATRIX_DATE[2,0] := ANY_TO_DATE(1445385600 + MATRIX_STRUCTURE_NON_RETAIN.MATRIX_DINT[2,0] * 86400);
    MATRIX_STRUCTURE_NON_RETAIN.MATRIX_DATE[2,1] := ANY_TO_DATE(1445385600 + MATRIX_STRUCTURE_NON_RETAIN.MATRIX_DINT[2,1] * 86400);
    MATRIX_STRUCTURE_NON_RETAIN.MATRIX_DATE[2,2] := ANY_TO_DATE(1445385600 + MATRIX_STRUCTURE_NON_RETAIN.MATRIX_DINT[2,2] * 86400);
    MATRIX_STRUCTURE_NON_RETAIN.MATRIX_DATE[2,3] := ANY_TO_DATE(1445385600 + MATRIX_STRUCTURE_NON_RETAIN.MATRIX_DINT[2,3] * 86400);
    MATRIX_STRUCTURE_NON_RETAIN.MATRIX_DATE[2,4] := ANY_TO_DATE(1445385600 + MATRIX_STRUCTURE_NON_RETAIN.MATRIX_DINT[2,4] * 86400);
    MATRIX_STRUCTURE_NON_RETAIN.MATRIX_DATE[2,5] := ANY_TO_DATE(1445385600 + MATRIX_STRUCTURE_NON_RETAIN.MATRIX_DINT[2,5] * 86400);
    MATRIX_STRUCTURE_NON_RETAIN.MATRIX_DATE[2,6] := ANY_TO_DATE(1445385600 + MATRIX_STRUCTURE_NON_RETAIN.MATRIX_DINT[2,6] * 86400);
    MATRIX_STRUCTURE_NON_RETAIN.MATRIX_DATE[2,7] := ANY_TO_DATE(1445385600 + MATRIX_STRUCTURE_NON_RETAIN.MATRIX_DINT[2,7] * 86400);
    MATRIX_STRUCTURE_NON_RETAIN.MATRIX_DATE[2,8] := ANY_TO_DATE(1445385600 + MATRIX_STRUCTURE_NON_RETAIN.MATRIX_DINT[2,8] * 86400);
    MATRIX_STRUCTURE_NON_RETAIN.MATRIX_DATE[2,9] := ANY_TO_DATE(1445385600 + MATRIX_STRUCTURE_NON_RETAIN.MATRIX_DINT[2,9] * 86400);

    MATRIX_STRUCTURE_NON_RETAIN.MATRIX_DATE[3,0] := ANY_TO_DATE(1445385600 + MATRIX_STRUCTURE_NON_RETAIN.MATRIX_DINT[3,0] * 86400);
    MATRIX_STRUCTURE_NON_RETAIN.MATRIX_DATE[3,1] := ANY_TO_DATE(1445385600 + MATRIX_STRUCTURE_NON_RETAIN.MATRIX_DINT[3,1] * 86400);
    MATRIX_STRUCTURE_NON_RETAIN.MATRIX_DATE[3,2] := ANY_TO_DATE(1445385600 + MATRIX_STRUCTURE_NON_RETAIN.MATRIX_DINT[3,2] * 86400);
    MATRIX_STRUCTURE_NON_RETAIN.MATRIX_DATE[3,3] := ANY_TO_DATE(1445385600 + MATRIX_STRUCTURE_NON_RETAIN.MATRIX_DINT[3,3] * 86400);
    MATRIX_STRUCTURE_NON_RETAIN.MATRIX_DATE[3,4] := ANY_TO_DATE(1445385600 + MATRIX_STRUCTURE_NON_RETAIN.MATRIX_DINT[3,4] * 86400);
    MATRIX_STRUCTURE_NON_RETAIN.MATRIX_DATE[3,5] := ANY_TO_DATE(1445385600 + MATRIX_STRUCTURE_NON_RETAIN.MATRIX_DINT[3,5] * 86400);
    MATRIX_STRUCTURE_NON_RETAIN.MATRIX_DATE[3,6] := ANY_TO_DATE(1445385600 + MATRIX_STRUCTURE_NON_RETAIN.MATRIX_DINT[3,6] * 86400);
    MATRIX_STRUCTURE_NON_RETAIN.MATRIX_DATE[3,7] := ANY_TO_DATE(1445385600 + MATRIX_STRUCTURE_NON_RETAIN.MATRIX_DINT[3,7] * 86400);
    MATRIX_STRUCTURE_NON_RETAIN.MATRIX_DATE[3,8] := ANY_TO_DATE(1445385600 + MATRIX_STRUCTURE_NON_RETAIN.MATRIX_DINT[3,8] * 86400);
    MATRIX_STRUCTURE_NON_RETAIN.MATRIX_DATE[3,9] := ANY_TO_DATE(1445385600 + MATRIX_STRUCTURE_NON_RETAIN.MATRIX_DINT[3,9] * 86400);

    MATRIX_STRUCTURE_NON_RETAIN.MATRIX_DATE[4,0] := ANY_TO_DATE(1445385600 + MATRIX_STRUCTURE_NON_RETAIN.MATRIX_DINT[4,0] * 86400);
    MATRIX_STRUCTURE_NON_RETAIN.MATRIX_DATE[4,1] := ANY_TO_DATE(1445385600 + MATRIX_STRUCTURE_NON_RETAIN.MATRIX_DINT[4,1] * 86400);
    MATRIX_STRUCTURE_NON_RETAIN.MATRIX_DATE[4,2] := ANY_TO_DATE(1445385600 + MATRIX_STRUCTURE_NON_RETAIN.MATRIX_DINT[4,2] * 86400);
    MATRIX_STRUCTURE_NON_RETAIN.MATRIX_DATE[4,3] := ANY_TO_DATE(1445385600 + MATRIX_STRUCTURE_NON_RETAIN.MATRIX_DINT[4,3] * 86400);
    MATRIX_STRUCTURE_NON_RETAIN.MATRIX_DATE[4,4] := ANY_TO_DATE(1445385600 + MATRIX_STRUCTURE_NON_RETAIN.MATRIX_DINT[4,4] * 86400);
    MATRIX_STRUCTURE_NON_RETAIN.MATRIX_DATE[4,5] := ANY_TO_DATE(1445385600 + MATRIX_STRUCTURE_NON_RETAIN.MATRIX_DINT[4,5] * 86400);
    MATRIX_STRUCTURE_NON_RETAIN.MATRIX_DATE[4,6] := ANY_TO_DATE(1445385600 + MATRIX_STRUCTURE_NON_RETAIN.MATRIX_DINT[4,6] * 86400);
    MATRIX_STRUCTURE_NON_RETAIN.MATRIX_DATE[4,7] := ANY_TO_DATE(1445385600 + MATRIX_STRUCTURE_NON_RETAIN.MATRIX_DINT[4,7] * 86400);
    MATRIX_STRUCTURE_NON_RETAIN.MATRIX_DATE[4,8] := ANY_TO_DATE(1445385600 + MATRIX_STRUCTURE_NON_RETAIN.MATRIX_DINT[4,8] * 86400);
    MATRIX_STRUCTURE_NON_RETAIN.MATRIX_DATE[4,9] := ANY_TO_DATE(1445385600 + MATRIX_STRUCTURE_NON_RETAIN.MATRIX_DINT[4,9] * 86400);

    MATRIX_STRUCTURE_NON_RETAIN.MATRIX_DATE[5,0] := ANY_TO_DATE(1445385600 + MATRIX_STRUCTURE_NON_RETAIN.MATRIX_DINT[5,0] * 86400);
    MATRIX_STRUCTURE_NON_RETAIN.MATRIX_DATE[5,1] := ANY_TO_DATE(1445385600 + MATRIX_STRUCTURE_NON_RETAIN.MATRIX_DINT[5,1] * 86400);
    MATRIX_STRUCTURE_NON_RETAIN.MATRIX_DATE[5,2] := ANY_TO_DATE(1445385600 + MATRIX_STRUCTURE_NON_RETAIN.MATRIX_DINT[5,2] * 86400);
    MATRIX_STRUCTURE_NON_RETAIN.MATRIX_DATE[5,3] := ANY_TO_DATE(1445385600 + MATRIX_STRUCTURE_NON_RETAIN.MATRIX_DINT[5,3] * 86400);
    MATRIX_STRUCTURE_NON_RETAIN.MATRIX_DATE[5,4] := ANY_TO_DATE(1445385600 + MATRIX_STRUCTURE_NON_RETAIN.MATRIX_DINT[5,4] * 86400);
    MATRIX_STRUCTURE_NON_RETAIN.MATRIX_DATE[5,5] := ANY_TO_DATE(1445385600 + MATRIX_STRUCTURE_NON_RETAIN.MATRIX_DINT[5,5] * 86400);
    MATRIX_STRUCTURE_NON_RETAIN.MATRIX_DATE[5,6] := ANY_TO_DATE(1445385600 + MATRIX_STRUCTURE_NON_RETAIN.MATRIX_DINT[5,6] * 86400);
    MATRIX_STRUCTURE_NON_RETAIN.MATRIX_DATE[5,7] := ANY_TO_DATE(1445385600 + MATRIX_STRUCTURE_NON_RETAIN.MATRIX_DINT[5,7] * 86400);
    MATRIX_STRUCTURE_NON_RETAIN.MATRIX_DATE[5,8] := ANY_TO_DATE(1445385600 + MATRIX_STRUCTURE_NON_RETAIN.MATRIX_DINT[5,8] * 86400);
    MATRIX_STRUCTURE_NON_RETAIN.MATRIX_DATE[5,9] := ANY_TO_DATE(1445385600 + MATRIX_STRUCTURE_NON_RETAIN.MATRIX_DINT[5,9] * 86400);

    MATRIX_STRUCTURE_NON_RETAIN.MATRIX_DATE[6,0] := ANY_TO_DATE(1445385600 + MATRIX_STRUCTURE_NON_RETAIN.MATRIX_DINT[6,0] * 86400);
    MATRIX_STRUCTURE_NON_RETAIN.MATRIX_DATE[6,1] := ANY_TO_DATE(1445385600 + MATRIX_STRUCTURE_NON_RETAIN.MATRIX_DINT[6,1] * 86400);
    MATRIX_STRUCTURE_NON_RETAIN.MATRIX_DATE[6,2] := ANY_TO_DATE(1445385600 + MATRIX_STRUCTURE_NON_RETAIN.MATRIX_DINT[6,2] * 86400);
    MATRIX_STRUCTURE_NON_RETAIN.MATRIX_DATE[6,3] := ANY_TO_DATE(1445385600 + MATRIX_STRUCTURE_NON_RETAIN.MATRIX_DINT[6,3] * 86400);
    MATRIX_STRUCTURE_NON_RETAIN.MATRIX_DATE[6,4] := ANY_TO_DATE(1445385600 + MATRIX_STRUCTURE_NON_RETAIN.MATRIX_DINT[6,4] * 86400);
    MATRIX_STRUCTURE_NON_RETAIN.MATRIX_DATE[6,5] := ANY_TO_DATE(1445385600 + MATRIX_STRUCTURE_NON_RETAIN.MATRIX_DINT[6,5] * 86400);
    MATRIX_STRUCTURE_NON_RETAIN.MATRIX_DATE[6,6] := ANY_TO_DATE(1445385600 + MATRIX_STRUCTURE_NON_RETAIN.MATRIX_DINT[6,6] * 86400);
    MATRIX_STRUCTURE_NON_RETAIN.MATRIX_DATE[6,7] := ANY_TO_DATE(1445385600 + MATRIX_STRUCTURE_NON_RETAIN.MATRIX_DINT[6,7] * 86400);
    MATRIX_STRUCTURE_NON_RETAIN.MATRIX_DATE[6,8] := ANY_TO_DATE(1445385600 + MATRIX_STRUCTURE_NON_RETAIN.MATRIX_DINT[6,8] * 86400);
    MATRIX_STRUCTURE_NON_RETAIN.MATRIX_DATE[6,9] := ANY_TO_DATE(1445385600 + MATRIX_STRUCTURE_NON_RETAIN.MATRIX_DINT[6,9] * 86400);

    MATRIX_STRUCTURE_NON_RETAIN.MATRIX_DATE[7,0] := MATRIX_STRUCTURE_NON_RETAIN.MATRIX_DATE[6,0];
    MATRIX_STRUCTURE_NON_RETAIN.MATRIX_DATE[7,1] := MATRIX_STRUCTURE_NON_RETAIN.MATRIX_DATE[6,1];
    MATRIX_STRUCTURE_NON_RETAIN.MATRIX_DATE[7,2] := MATRIX_STRUCTURE_NON_RETAIN.MATRIX_DATE[6,2];
    MATRIX_STRUCTURE_NON_RETAIN.MATRIX_DATE[7,3] := MATRIX_STRUCTURE_NON_RETAIN.MATRIX_DATE[6,3];
    MATRIX_STRUCTURE_NON_RETAIN.MATRIX_DATE[7,4] := MATRIX_STRUCTURE_NON_RETAIN.MATRIX_DATE[6,4];
    MATRIX_STRUCTURE_NON_RETAIN.MATRIX_DATE[7,5] := MATRIX_STRUCTURE_NON_RETAIN.MATRIX_DATE[6,5];
    MATRIX_STRUCTURE_NON_RETAIN.MATRIX_DATE[7,6] := MATRIX_STRUCTURE_NON_RETAIN.MATRIX_DATE[6,6];
    MATRIX_STRUCTURE_NON_RETAIN.MATRIX_DATE[7,7] := MATRIX_STRUCTURE_NON_RETAIN.MATRIX_DATE[6,7];
    MATRIX_STRUCTURE_NON_RETAIN.MATRIX_DATE[7,8] := MATRIX_STRUCTURE_NON_RETAIN.MATRIX_DATE[6,8];
    MATRIX_STRUCTURE_NON_RETAIN.MATRIX_DATE[7,9] := MATRIX_STRUCTURE_NON_RETAIN.MATRIX_DATE[6,9];

    MATRIX_STRUCTURE_NON_RETAIN.MATRIX_DINT[0,0] := MATRIX_STRUCTURE_NON_RETAIN.MATRIX_DINT[0,0] + 1;
    MATRIX_STRUCTURE_NON_RETAIN.MATRIX_DINT[0,1] := MATRIX_STRUCTURE_NON_RETAIN.MATRIX_DINT[0,1] + 1;
    MATRIX_STRUCTURE_NON_RETAIN.MATRIX_DINT[0,2] := MATRIX_STRUCTURE_NON_RETAIN.MATRIX_DINT[0,2] + 1;
    MATRIX_STRUCTURE_NON_RETAIN.MATRIX_DINT[0,3] := MATRIX_STRUCTURE_NON_RETAIN.MATRIX_DINT[0,3] + 1;
    MATRIX_STRUCTURE_NON_RETAIN.MATRIX_DINT[0,4] := MATRIX_STRUCTURE_NON_RETAIN.MATRIX_DINT[0,4] + 1;
    MATRIX_STRUCTURE_NON_RETAIN.MATRIX_DINT[0,5] := MATRIX_STRUCTURE_NON_RETAIN.MATRIX_DINT[0,5] + 1;
    MATRIX_STRUCTURE_NON_RETAIN.MATRIX_DINT[0,6] := MATRIX_STRUCTURE_NON_RETAIN.MATRIX_DINT[0,6] + 1;
    MATRIX_STRUCTURE_NON_RETAIN.MATRIX_DINT[0,7] := MATRIX_STRUCTURE_NON_RETAIN.MATRIX_DINT[0,7] + 1;
    MATRIX_STRUCTURE_NON_RETAIN.MATRIX_DINT[0,8] := MATRIX_STRUCTURE_NON_RETAIN.MATRIX_DINT[0,6];
    MATRIX_STRUCTURE_NON_RETAIN.MATRIX_DINT[0,9] := MATRIX_STRUCTURE_NON_RETAIN.MATRIX_DINT[0,7];

    MATRIX_STRUCTURE_NON_RETAIN.MATRIX_DINT[1,0] := MATRIX_STRUCTURE_NON_RETAIN.MATRIX_DINT[1,0] + 1;
    MATRIX_STRUCTURE_NON_RETAIN.MATRIX_DINT[1,1] := MATRIX_STRUCTURE_NON_RETAIN.MATRIX_DINT[1,1] + 1;
    MATRIX_STRUCTURE_NON_RETAIN.MATRIX_DINT[1,2] := MATRIX_STRUCTURE_NON_RETAIN.MATRIX_DINT[1,2] + 1;
    MATRIX_STRUCTURE_NON_RETAIN.MATRIX_DINT[1,3] := MATRIX_STRUCTURE_NON_RETAIN.MATRIX_DINT[1,3] + 1;
    MATRIX_STRUCTURE_NON_RETAIN.MATRIX_DINT[1,4] := MATRIX_STRUCTURE_NON_RETAIN.MATRIX_DINT[1,4] + 1;
    MATRIX_STRUCTURE_NON_RETAIN.MATRIX_DINT[1,5] := MATRIX_STRUCTURE_NON_RETAIN.MATRIX_DINT[1,5] + 1;
    MATRIX_STRUCTURE_NON_RETAIN.MATRIX_DINT[1,6] := MATRIX_STRUCTURE_NON_RETAIN.MATRIX_DINT[1,6] + 1;
    MATRIX_STRUCTURE_NON_RETAIN.MATRIX_DINT[1,7] := MATRIX_STRUCTURE_NON_RETAIN.MATRIX_DINT[1,7] + 1;
    MATRIX_STRUCTURE_NON_RETAIN.MATRIX_DINT[1,8] := MATRIX_STRUCTURE_NON_RETAIN.MATRIX_DINT[1,8];
    MATRIX_STRUCTURE_NON_RETAIN.MATRIX_DINT[1,9] := MATRIX_STRUCTURE_NON_RETAIN.MATRIX_DINT[1,9];

    MATRIX_STRUCTURE_NON_RETAIN.MATRIX_DINT[2,0] := MATRIX_STRUCTURE_NON_RETAIN.MATRIX_DINT[2,0] + 1;
    MATRIX_STRUCTURE_NON_RETAIN.MATRIX_DINT[2,1] := MATRIX_STRUCTURE_NON_RETAIN.MATRIX_DINT[2,1] + 1;
    MATRIX_STRUCTURE_NON_RETAIN.MATRIX_DINT[2,2] := MATRIX_STRUCTURE_NON_RETAIN.MATRIX_DINT[2,2] + 1;
    MATRIX_STRUCTURE_NON_RETAIN.MATRIX_DINT[2,3] := MATRIX_STRUCTURE_NON_RETAIN.MATRIX_DINT[2,3] + 1;
    MATRIX_STRUCTURE_NON_RETAIN.MATRIX_DINT[2,4] := MATRIX_STRUCTURE_NON_RETAIN.MATRIX_DINT[2,4] + 1;
    MATRIX_STRUCTURE_NON_RETAIN.MATRIX_DINT[2,5] := MATRIX_STRUCTURE_NON_RETAIN.MATRIX_DINT[2,5] + 1;
    MATRIX_STRUCTURE_NON_RETAIN.MATRIX_DINT[2,6] := MATRIX_STRUCTURE_NON_RETAIN.MATRIX_DINT[2,6] + 1;
    MATRIX_STRUCTURE_NON_RETAIN.MATRIX_DINT[2,7] := MATRIX_STRUCTURE_NON_RETAIN.MATRIX_DINT[2,7] + 1;
    MATRIX_STRUCTURE_NON_RETAIN.MATRIX_DINT[2,8] := MATRIX_STRUCTURE_NON_RETAIN.MATRIX_DINT[2,8] + 1;
    MATRIX_STRUCTURE_NON_RETAIN.MATRIX_DINT[2,9] := MATRIX_STRUCTURE_NON_RETAIN.MATRIX_DINT[2,9] + 1;

    MATRIX_STRUCTURE_NON_RETAIN.MATRIX_DINT[3,0] := MATRIX_STRUCTURE_NON_RETAIN.MATRIX_DINT[3,0] + 1;
    MATRIX_STRUCTURE_NON_RETAIN.MATRIX_DINT[3,1] := MATRIX_STRUCTURE_NON_RETAIN.MATRIX_DINT[3,1] + 1;
    MATRIX_STRUCTURE_NON_RETAIN.MATRIX_DINT[3,2] := MATRIX_STRUCTURE_NON_RETAIN.MATRIX_DINT[3,2] + 1;
    MATRIX_STRUCTURE_NON_RETAIN.MATRIX_DINT[3,3] := MATRIX_STRUCTURE_NON_RETAIN.MATRIX_DINT[3,3] + 1;
    MATRIX_STRUCTURE_NON_RETAIN.MATRIX_DINT[3,4] := MATRIX_STRUCTURE_NON_RETAIN.MATRIX_DINT[3,4] + 1;
    MATRIX_STRUCTURE_NON_RETAIN.MATRIX_DINT[3,5] := MATRIX_STRUCTURE_NON_RETAIN.MATRIX_DINT[3,5] + 1;
    MATRIX_STRUCTURE_NON_RETAIN.MATRIX_DINT[3,6] := MATRIX_STRUCTURE_NON_RETAIN.MATRIX_DINT[3,6] + 1;
    MATRIX_STRUCTURE_NON_RETAIN.MATRIX_DINT[3,7] := MATRIX_STRUCTURE_NON_RETAIN.MATRIX_DINT[3,7] + 1;
    MATRIX_STRUCTURE_NON_RETAIN.MATRIX_DINT[3,8] := MATRIX_STRUCTURE_NON_RETAIN.MATRIX_DINT[3,8] + 1;
    MATRIX_STRUCTURE_NON_RETAIN.MATRIX_DINT[3,9] := MATRIX_STRUCTURE_NON_RETAIN.MATRIX_DINT[3,9] + 1;

    MATRIX_STRUCTURE_NON_RETAIN.MATRIX_DINT[4,0] := MATRIX_STRUCTURE_NON_RETAIN.MATRIX_DINT[4,0] + 1;
    MATRIX_STRUCTURE_NON_RETAIN.MATRIX_DINT[4,1] := MATRIX_STRUCTURE_NON_RETAIN.MATRIX_DINT[4,1] + 1;
    MATRIX_STRUCTURE_NON_RETAIN.MATRIX_DINT[4,2] := MATRIX_STRUCTURE_NON_RETAIN.MATRIX_DINT[4,2] + 1;
    MATRIX_STRUCTURE_NON_RETAIN.MATRIX_DINT[4,3] := MATRIX_STRUCTURE_NON_RETAIN.MATRIX_DINT[4,3] + 1;
    MATRIX_STRUCTURE_NON_RETAIN.MATRIX_DINT[4,4] := MATRIX_STRUCTURE_NON_RETAIN.MATRIX_DINT[4,4] + 1;
    MATRIX_STRUCTURE_NON_RETAIN.MATRIX_DINT[4,5] := MATRIX_STRUCTURE_NON_RETAIN.MATRIX_DINT[4,5] + 1;
    MATRIX_STRUCTURE_NON_RETAIN.MATRIX_DINT[4,6] := MATRIX_STRUCTURE_NON_RETAIN.MATRIX_DINT[4,6] + 1;
    MATRIX_STRUCTURE_NON_RETAIN.MATRIX_DINT[4,7] := MATRIX_STRUCTURE_NON_RETAIN.MATRIX_DINT[4,7] + 1;
    MATRIX_STRUCTURE_NON_RETAIN.MATRIX_DINT[4,8] := MATRIX_STRUCTURE_NON_RETAIN.MATRIX_DINT[4,8] + 1;
    MATRIX_STRUCTURE_NON_RETAIN.MATRIX_DINT[4,9] := MATRIX_STRUCTURE_NON_RETAIN.MATRIX_DINT[4,9] + 1;

    MATRIX_STRUCTURE_NON_RETAIN.MATRIX_DINT[5,0] := MATRIX_STRUCTURE_NON_RETAIN.MATRIX_DINT[5,0] + 1;
    MATRIX_STRUCTURE_NON_RETAIN.MATRIX_DINT[5,1] := MATRIX_STRUCTURE_NON_RETAIN.MATRIX_DINT[5,1] + 1;
    MATRIX_STRUCTURE_NON_RETAIN.MATRIX_DINT[5,2] := MATRIX_STRUCTURE_NON_RETAIN.MATRIX_DINT[5,2] + 1;
    MATRIX_STRUCTURE_NON_RETAIN.MATRIX_DINT[5,3] := MATRIX_STRUCTURE_NON_RETAIN.MATRIX_DINT[5,3] + 1;
    MATRIX_STRUCTURE_NON_RETAIN.MATRIX_DINT[5,4] := MATRIX_STRUCTURE_NON_RETAIN.MATRIX_DINT[5,4] + 1;
    MATRIX_STRUCTURE_NON_RETAIN.MATRIX_DINT[5,5] := MATRIX_STRUCTURE_NON_RETAIN.MATRIX_DINT[5,5] + 1;
    MATRIX_STRUCTURE_NON_RETAIN.MATRIX_DINT[5,6] := MATRIX_STRUCTURE_NON_RETAIN.MATRIX_DINT[5,6] + 1;
    MATRIX_STRUCTURE_NON_RETAIN.MATRIX_DINT[5,7] := MATRIX_STRUCTURE_NON_RETAIN.MATRIX_DINT[5,7] + 1;
    MATRIX_STRUCTURE_NON_RETAIN.MATRIX_DINT[5,8] := MATRIX_STRUCTURE_NON_RETAIN.MATRIX_DINT[5,8] + 1;
    MATRIX_STRUCTURE_NON_RETAIN.MATRIX_DINT[5,9] := MATRIX_STRUCTURE_NON_RETAIN.MATRIX_DINT[5,9] + 1;

    MATRIX_STRUCTURE_NON_RETAIN.MATRIX_DINT[6,0] := MATRIX_STRUCTURE_NON_RETAIN.MATRIX_DINT[6,0] + 1;
    MATRIX_STRUCTURE_NON_RETAIN.MATRIX_DINT[6,1] := MATRIX_STRUCTURE_NON_RETAIN.MATRIX_DINT[6,1] + 1;
    MATRIX_STRUCTURE_NON_RETAIN.MATRIX_DINT[6,2] := MATRIX_STRUCTURE_NON_RETAIN.MATRIX_DINT[6,2] + 1;
    MATRIX_STRUCTURE_NON_RETAIN.MATRIX_DINT[6,3] := MATRIX_STRUCTURE_NON_RETAIN.MATRIX_DINT[6,3] + 1;
    MATRIX_STRUCTURE_NON_RETAIN.MATRIX_DINT[6,4] := MATRIX_STRUCTURE_NON_RETAIN.MATRIX_DINT[6,4] + 1;
    MATRIX_STRUCTURE_NON_RETAIN.MATRIX_DINT[6,5] := MATRIX_STRUCTURE_NON_RETAIN.MATRIX_DINT[6,5] + 1;
    MATRIX_STRUCTURE_NON_RETAIN.MATRIX_DINT[6,6] := MATRIX_STRUCTURE_NON_RETAIN.MATRIX_DINT[6,6] + 1;
    MATRIX_STRUCTURE_NON_RETAIN.MATRIX_DINT[6,7] := MATRIX_STRUCTURE_NON_RETAIN.MATRIX_DINT[6,7] + 1;
    MATRIX_STRUCTURE_NON_RETAIN.MATRIX_DINT[6,8] := MATRIX_STRUCTURE_NON_RETAIN.MATRIX_DINT[6,8] + 1;
    MATRIX_STRUCTURE_NON_RETAIN.MATRIX_DINT[6,9] := MATRIX_STRUCTURE_NON_RETAIN.MATRIX_DINT[6,9] + 1;

    MATRIX_STRUCTURE_NON_RETAIN.MATRIX_DINT[7,0] := MATRIX_STRUCTURE_NON_RETAIN.MATRIX_DINT[6,0];
    MATRIX_STRUCTURE_NON_RETAIN.MATRIX_DINT[7,1] := MATRIX_STRUCTURE_NON_RETAIN.MATRIX_DINT[6,1];
    MATRIX_STRUCTURE_NON_RETAIN.MATRIX_DINT[7,2] := MATRIX_STRUCTURE_NON_RETAIN.MATRIX_DINT[6,2];
    MATRIX_STRUCTURE_NON_RETAIN.MATRIX_DINT[7,3] := MATRIX_STRUCTURE_NON_RETAIN.MATRIX_DINT[6,3];
    MATRIX_STRUCTURE_NON_RETAIN.MATRIX_DINT[7,4] := MATRIX_STRUCTURE_NON_RETAIN.MATRIX_DINT[6,4];
    MATRIX_STRUCTURE_NON_RETAIN.MATRIX_DINT[7,5] := MATRIX_STRUCTURE_NON_RETAIN.MATRIX_DINT[6,5];
    MATRIX_STRUCTURE_NON_RETAIN.MATRIX_DINT[7,6] := MATRIX_STRUCTURE_NON_RETAIN.MATRIX_DINT[6,6];
    MATRIX_STRUCTURE_NON_RETAIN.MATRIX_DINT[7,7] := MATRIX_STRUCTURE_NON_RETAIN.MATRIX_DINT[6,7];
    MATRIX_STRUCTURE_NON_RETAIN.MATRIX_DINT[7,8] := MATRIX_STRUCTURE_NON_RETAIN.MATRIX_DINT[6,8];
    MATRIX_STRUCTURE_NON_RETAIN.MATRIX_DINT[7,9] := MATRIX_STRUCTURE_NON_RETAIN.MATRIX_DINT[6,9];

    MATRIX_STRUCTURE_NON_RETAIN.MATRIX_DWORD[0,0] := MATRIX_STRUCTURE_NON_RETAIN.MATRIX_DWORD[0,0] + 1;
    MATRIX_STRUCTURE_NON_RETAIN.MATRIX_DWORD[0,1] := MATRIX_STRUCTURE_NON_RETAIN.MATRIX_DWORD[0,1] + 1;
    MATRIX_STRUCTURE_NON_RETAIN.MATRIX_DWORD[0,2] := MATRIX_STRUCTURE_NON_RETAIN.MATRIX_DWORD[0,2] + 1;
    MATRIX_STRUCTURE_NON_RETAIN.MATRIX_DWORD[0,3] := MATRIX_STRUCTURE_NON_RETAIN.MATRIX_DWORD[0,3] + 1;
    MATRIX_STRUCTURE_NON_RETAIN.MATRIX_DWORD[0,4] := MATRIX_STRUCTURE_NON_RETAIN.MATRIX_DWORD[0,4] + 1;
    MATRIX_STRUCTURE_NON_RETAIN.MATRIX_DWORD[0,5] := MATRIX_STRUCTURE_NON_RETAIN.MATRIX_DWORD[0,5] + 1;
    MATRIX_STRUCTURE_NON_RETAIN.MATRIX_DWORD[0,6] := MATRIX_STRUCTURE_NON_RETAIN.MATRIX_DWORD[0,6] + 1;
    MATRIX_STRUCTURE_NON_RETAIN.MATRIX_DWORD[0,7] := MATRIX_STRUCTURE_NON_RETAIN.MATRIX_DWORD[0,7] + 1;
    MATRIX_STRUCTURE_NON_RETAIN.MATRIX_DWORD[0,8] := MATRIX_STRUCTURE_NON_RETAIN.MATRIX_DWORD[0,6];
    MATRIX_STRUCTURE_NON_RETAIN.MATRIX_DWORD[0,9] := MATRIX_STRUCTURE_NON_RETAIN.MATRIX_DWORD[0,7];

    MATRIX_STRUCTURE_NON_RETAIN.MATRIX_DWORD[1,0] := MATRIX_STRUCTURE_NON_RETAIN.MATRIX_DWORD[1,0] + 1;
    MATRIX_STRUCTURE_NON_RETAIN.MATRIX_DWORD[1,1] := MATRIX_STRUCTURE_NON_RETAIN.MATRIX_DWORD[1,1] + 1;
    MATRIX_STRUCTURE_NON_RETAIN.MATRIX_DWORD[1,2] := MATRIX_STRUCTURE_NON_RETAIN.MATRIX_DWORD[1,2] + 1;
    MATRIX_STRUCTURE_NON_RETAIN.MATRIX_DWORD[1,3] := MATRIX_STRUCTURE_NON_RETAIN.MATRIX_DWORD[1,3] + 1;
    MATRIX_STRUCTURE_NON_RETAIN.MATRIX_DWORD[1,4] := MATRIX_STRUCTURE_NON_RETAIN.MATRIX_DWORD[1,4] + 1;
    MATRIX_STRUCTURE_NON_RETAIN.MATRIX_DWORD[1,5] := MATRIX_STRUCTURE_NON_RETAIN.MATRIX_DWORD[1,5] + 1;
    MATRIX_STRUCTURE_NON_RETAIN.MATRIX_DWORD[1,6] := MATRIX_STRUCTURE_NON_RETAIN.MATRIX_DWORD[1,6] + 1;
    MATRIX_STRUCTURE_NON_RETAIN.MATRIX_DWORD[1,7] := MATRIX_STRUCTURE_NON_RETAIN.MATRIX_DWORD[1,7] + 1;
    MATRIX_STRUCTURE_NON_RETAIN.MATRIX_DWORD[1,8] := MATRIX_STRUCTURE_NON_RETAIN.MATRIX_DWORD[1,6];
    MATRIX_STRUCTURE_NON_RETAIN.MATRIX_DWORD[1,9] := MATRIX_STRUCTURE_NON_RETAIN.MATRIX_DWORD[1,7];

    MATRIX_STRUCTURE_NON_RETAIN.MATRIX_DWORD[2,0] := MATRIX_STRUCTURE_NON_RETAIN.MATRIX_DWORD[2,0] + 1;
    MATRIX_STRUCTURE_NON_RETAIN.MATRIX_DWORD[2,1] := MATRIX_STRUCTURE_NON_RETAIN.MATRIX_DWORD[2,1] + 1;
    MATRIX_STRUCTURE_NON_RETAIN.MATRIX_DWORD[2,2] := MATRIX_STRUCTURE_NON_RETAIN.MATRIX_DWORD[2,2] + 1;
    MATRIX_STRUCTURE_NON_RETAIN.MATRIX_DWORD[2,3] := MATRIX_STRUCTURE_NON_RETAIN.MATRIX_DWORD[2,3] + 1;
    MATRIX_STRUCTURE_NON_RETAIN.MATRIX_DWORD[2,4] := MATRIX_STRUCTURE_NON_RETAIN.MATRIX_DWORD[2,4] + 1;
    MATRIX_STRUCTURE_NON_RETAIN.MATRIX_DWORD[2,5] := MATRIX_STRUCTURE_NON_RETAIN.MATRIX_DWORD[2,5] + 1;
    MATRIX_STRUCTURE_NON_RETAIN.MATRIX_DWORD[2,6] := MATRIX_STRUCTURE_NON_RETAIN.MATRIX_DWORD[2,6] + 1;
    MATRIX_STRUCTURE_NON_RETAIN.MATRIX_DWORD[2,7] := MATRIX_STRUCTURE_NON_RETAIN.MATRIX_DWORD[2,7] + 1;
    MATRIX_STRUCTURE_NON_RETAIN.MATRIX_DWORD[2,8] := MATRIX_STRUCTURE_NON_RETAIN.MATRIX_DWORD[2,8] + 1;
    MATRIX_STRUCTURE_NON_RETAIN.MATRIX_DWORD[2,9] := MATRIX_STRUCTURE_NON_RETAIN.MATRIX_DWORD[2,9] + 1;

    MATRIX_STRUCTURE_NON_RETAIN.MATRIX_DWORD[3,0] := MATRIX_STRUCTURE_NON_RETAIN.MATRIX_DWORD[3,0] + 1;
    MATRIX_STRUCTURE_NON_RETAIN.MATRIX_DWORD[3,1] := MATRIX_STRUCTURE_NON_RETAIN.MATRIX_DWORD[3,1] + 1;
    MATRIX_STRUCTURE_NON_RETAIN.MATRIX_DWORD[3,2] := MATRIX_STRUCTURE_NON_RETAIN.MATRIX_DWORD[3,2] + 1;
    MATRIX_STRUCTURE_NON_RETAIN.MATRIX_DWORD[3,3] := MATRIX_STRUCTURE_NON_RETAIN.MATRIX_DWORD[3,3] + 1;
    MATRIX_STRUCTURE_NON_RETAIN.MATRIX_DWORD[3,4] := MATRIX_STRUCTURE_NON_RETAIN.MATRIX_DWORD[3,4] + 1;
    MATRIX_STRUCTURE_NON_RETAIN.MATRIX_DWORD[3,5] := MATRIX_STRUCTURE_NON_RETAIN.MATRIX_DWORD[3,5] + 1;
    MATRIX_STRUCTURE_NON_RETAIN.MATRIX_DWORD[3,6] := MATRIX_STRUCTURE_NON_RETAIN.MATRIX_DWORD[3,6] + 1;
    MATRIX_STRUCTURE_NON_RETAIN.MATRIX_DWORD[3,7] := MATRIX_STRUCTURE_NON_RETAIN.MATRIX_DWORD[3,7] + 1;
    MATRIX_STRUCTURE_NON_RETAIN.MATRIX_DWORD[3,8] := MATRIX_STRUCTURE_NON_RETAIN.MATRIX_DWORD[3,8] + 1;
    MATRIX_STRUCTURE_NON_RETAIN.MATRIX_DWORD[3,9] := MATRIX_STRUCTURE_NON_RETAIN.MATRIX_DWORD[3,9] + 1;

    MATRIX_STRUCTURE_NON_RETAIN.MATRIX_DWORD[4,0] := MATRIX_STRUCTURE_NON_RETAIN.MATRIX_DWORD[4,0] + 1;
    MATRIX_STRUCTURE_NON_RETAIN.MATRIX_DWORD[4,1] := MATRIX_STRUCTURE_NON_RETAIN.MATRIX_DWORD[4,1] + 1;
    MATRIX_STRUCTURE_NON_RETAIN.MATRIX_DWORD[4,2] := MATRIX_STRUCTURE_NON_RETAIN.MATRIX_DWORD[4,2] + 1;
    MATRIX_STRUCTURE_NON_RETAIN.MATRIX_DWORD[4,3] := MATRIX_STRUCTURE_NON_RETAIN.MATRIX_DWORD[4,3] + 1;
    MATRIX_STRUCTURE_NON_RETAIN.MATRIX_DWORD[4,4] := MATRIX_STRUCTURE_NON_RETAIN.MATRIX_DWORD[4,4] + 1;
    MATRIX_STRUCTURE_NON_RETAIN.MATRIX_DWORD[4,5] := MATRIX_STRUCTURE_NON_RETAIN.MATRIX_DWORD[4,5] + 1;
    MATRIX_STRUCTURE_NON_RETAIN.MATRIX_DWORD[4,6] := MATRIX_STRUCTURE_NON_RETAIN.MATRIX_DWORD[4,6] + 1;
    MATRIX_STRUCTURE_NON_RETAIN.MATRIX_DWORD[4,7] := MATRIX_STRUCTURE_NON_RETAIN.MATRIX_DWORD[4,7] + 1;
    MATRIX_STRUCTURE_NON_RETAIN.MATRIX_DWORD[4,8] := MATRIX_STRUCTURE_NON_RETAIN.MATRIX_DWORD[4,8] + 1;
    MATRIX_STRUCTURE_NON_RETAIN.MATRIX_DWORD[4,9] := MATRIX_STRUCTURE_NON_RETAIN.MATRIX_DWORD[4,9] + 1;

    MATRIX_STRUCTURE_NON_RETAIN.MATRIX_DWORD[5,0] := MATRIX_STRUCTURE_NON_RETAIN.MATRIX_DWORD[5,0] + 1;
    MATRIX_STRUCTURE_NON_RETAIN.MATRIX_DWORD[5,1] := MATRIX_STRUCTURE_NON_RETAIN.MATRIX_DWORD[5,1] + 1;
    MATRIX_STRUCTURE_NON_RETAIN.MATRIX_DWORD[5,2] := MATRIX_STRUCTURE_NON_RETAIN.MATRIX_DWORD[5,2] + 1;
    MATRIX_STRUCTURE_NON_RETAIN.MATRIX_DWORD[5,3] := MATRIX_STRUCTURE_NON_RETAIN.MATRIX_DWORD[5,3] + 1;
    MATRIX_STRUCTURE_NON_RETAIN.MATRIX_DWORD[5,4] := MATRIX_STRUCTURE_NON_RETAIN.MATRIX_DWORD[5,4] + 1;
    MATRIX_STRUCTURE_NON_RETAIN.MATRIX_DWORD[5,5] := MATRIX_STRUCTURE_NON_RETAIN.MATRIX_DWORD[5,5] + 1;
    MATRIX_STRUCTURE_NON_RETAIN.MATRIX_DWORD[5,6] := MATRIX_STRUCTURE_NON_RETAIN.MATRIX_DWORD[5,6] + 1;
    MATRIX_STRUCTURE_NON_RETAIN.MATRIX_DWORD[5,7] := MATRIX_STRUCTURE_NON_RETAIN.MATRIX_DWORD[5,7] + 1;
    MATRIX_STRUCTURE_NON_RETAIN.MATRIX_DWORD[5,8] := MATRIX_STRUCTURE_NON_RETAIN.MATRIX_DWORD[5,8] + 1;
    MATRIX_STRUCTURE_NON_RETAIN.MATRIX_DWORD[5,9] := MATRIX_STRUCTURE_NON_RETAIN.MATRIX_DWORD[5,9] + 1;

    MATRIX_STRUCTURE_NON_RETAIN.MATRIX_DWORD[6,0] := MATRIX_STRUCTURE_NON_RETAIN.MATRIX_DWORD[6,0] + 1;
    MATRIX_STRUCTURE_NON_RETAIN.MATRIX_DWORD[6,1] := MATRIX_STRUCTURE_NON_RETAIN.MATRIX_DWORD[6,1] + 1;
    MATRIX_STRUCTURE_NON_RETAIN.MATRIX_DWORD[6,2] := MATRIX_STRUCTURE_NON_RETAIN.MATRIX_DWORD[6,2] + 1;
    MATRIX_STRUCTURE_NON_RETAIN.MATRIX_DWORD[6,3] := MATRIX_STRUCTURE_NON_RETAIN.MATRIX_DWORD[6,3] + 1;
    MATRIX_STRUCTURE_NON_RETAIN.MATRIX_DWORD[6,4] := MATRIX_STRUCTURE_NON_RETAIN.MATRIX_DWORD[6,4] + 1;
    MATRIX_STRUCTURE_NON_RETAIN.MATRIX_DWORD[6,5] := MATRIX_STRUCTURE_NON_RETAIN.MATRIX_DWORD[6,5] + 1;
    MATRIX_STRUCTURE_NON_RETAIN.MATRIX_DWORD[6,6] := MATRIX_STRUCTURE_NON_RETAIN.MATRIX_DWORD[6,6] + 1;
    MATRIX_STRUCTURE_NON_RETAIN.MATRIX_DWORD[6,7] := MATRIX_STRUCTURE_NON_RETAIN.MATRIX_DWORD[6,7] + 1;
    MATRIX_STRUCTURE_NON_RETAIN.MATRIX_DWORD[6,8] := MATRIX_STRUCTURE_NON_RETAIN.MATRIX_DWORD[6,8] + 1;
    MATRIX_STRUCTURE_NON_RETAIN.MATRIX_DWORD[6,9] := MATRIX_STRUCTURE_NON_RETAIN.MATRIX_DWORD[6,9] + 1;

    MATRIX_STRUCTURE_NON_RETAIN.MATRIX_DWORD[7,0] := MATRIX_STRUCTURE_NON_RETAIN.MATRIX_DWORD[6,0];
    MATRIX_STRUCTURE_NON_RETAIN.MATRIX_DWORD[7,1] := MATRIX_STRUCTURE_NON_RETAIN.MATRIX_DWORD[6,1];
    MATRIX_STRUCTURE_NON_RETAIN.MATRIX_DWORD[7,2] := MATRIX_STRUCTURE_NON_RETAIN.MATRIX_DWORD[6,2];
    MATRIX_STRUCTURE_NON_RETAIN.MATRIX_DWORD[7,3] := MATRIX_STRUCTURE_NON_RETAIN.MATRIX_DWORD[6,3];
    MATRIX_STRUCTURE_NON_RETAIN.MATRIX_DWORD[7,4] := MATRIX_STRUCTURE_NON_RETAIN.MATRIX_DWORD[6,4];
    MATRIX_STRUCTURE_NON_RETAIN.MATRIX_DWORD[7,5] := MATRIX_STRUCTURE_NON_RETAIN.MATRIX_DWORD[6,5];
    MATRIX_STRUCTURE_NON_RETAIN.MATRIX_DWORD[7,6] := MATRIX_STRUCTURE_NON_RETAIN.MATRIX_DWORD[6,6];
    MATRIX_STRUCTURE_NON_RETAIN.MATRIX_DWORD[7,7] := MATRIX_STRUCTURE_NON_RETAIN.MATRIX_DWORD[6,7];
    MATRIX_STRUCTURE_NON_RETAIN.MATRIX_DWORD[7,8] := MATRIX_STRUCTURE_NON_RETAIN.MATRIX_DWORD[6,9];
    MATRIX_STRUCTURE_NON_RETAIN.MATRIX_DWORD[7,9] := MATRIX_STRUCTURE_NON_RETAIN.MATRIX_DWORD[6,9];

    MATRIX_STRUCTURE_NON_RETAIN.MATRIX_INT[0,0] := MATRIX_STRUCTURE_NON_RETAIN.MATRIX_INT[0,0] + 1;
    MATRIX_STRUCTURE_NON_RETAIN.MATRIX_INT[0,1] := MATRIX_STRUCTURE_NON_RETAIN.MATRIX_INT[0,1] + 1;
    MATRIX_STRUCTURE_NON_RETAIN.MATRIX_INT[0,2] := MATRIX_STRUCTURE_NON_RETAIN.MATRIX_INT[0,2] + 1;
    MATRIX_STRUCTURE_NON_RETAIN.MATRIX_INT[0,3] := MATRIX_STRUCTURE_NON_RETAIN.MATRIX_INT[0,3] + 1;
    MATRIX_STRUCTURE_NON_RETAIN.MATRIX_INT[0,4] := MATRIX_STRUCTURE_NON_RETAIN.MATRIX_INT[0,4] + 1;
    MATRIX_STRUCTURE_NON_RETAIN.MATRIX_INT[0,5] := MATRIX_STRUCTURE_NON_RETAIN.MATRIX_INT[0,5] + 1;
    MATRIX_STRUCTURE_NON_RETAIN.MATRIX_INT[0,6] := MATRIX_STRUCTURE_NON_RETAIN.MATRIX_INT[0,6] + 1;
    MATRIX_STRUCTURE_NON_RETAIN.MATRIX_INT[0,7] := MATRIX_STRUCTURE_NON_RETAIN.MATRIX_INT[0,7] + 1;
    MATRIX_STRUCTURE_NON_RETAIN.MATRIX_INT[0,8] := MATRIX_STRUCTURE_NON_RETAIN.MATRIX_INT[0,6];
    MATRIX_STRUCTURE_NON_RETAIN.MATRIX_INT[0,9] := MATRIX_STRUCTURE_NON_RETAIN.MATRIX_INT[0,7];

    MATRIX_STRUCTURE_NON_RETAIN.MATRIX_INT[1,0] := MATRIX_STRUCTURE_NON_RETAIN.MATRIX_INT[1,0] + 1;
    MATRIX_STRUCTURE_NON_RETAIN.MATRIX_INT[1,1] := MATRIX_STRUCTURE_NON_RETAIN.MATRIX_INT[1,1] + 1;
    MATRIX_STRUCTURE_NON_RETAIN.MATRIX_INT[1,2] := MATRIX_STRUCTURE_NON_RETAIN.MATRIX_INT[1,2] + 1;
    MATRIX_STRUCTURE_NON_RETAIN.MATRIX_INT[1,3] := MATRIX_STRUCTURE_NON_RETAIN.MATRIX_INT[1,3] + 1;
    MATRIX_STRUCTURE_NON_RETAIN.MATRIX_INT[1,4] := MATRIX_STRUCTURE_NON_RETAIN.MATRIX_INT[1,4] + 1;
    MATRIX_STRUCTURE_NON_RETAIN.MATRIX_INT[1,5] := MATRIX_STRUCTURE_NON_RETAIN.MATRIX_INT[1,5] + 1;
    MATRIX_STRUCTURE_NON_RETAIN.MATRIX_INT[1,6] := MATRIX_STRUCTURE_NON_RETAIN.MATRIX_INT[1,6] + 1;
    MATRIX_STRUCTURE_NON_RETAIN.MATRIX_INT[1,7] := MATRIX_STRUCTURE_NON_RETAIN.MATRIX_INT[1,7] + 1;
    MATRIX_STRUCTURE_NON_RETAIN.MATRIX_INT[1,8] := MATRIX_STRUCTURE_NON_RETAIN.MATRIX_INT[1,6];
    MATRIX_STRUCTURE_NON_RETAIN.MATRIX_INT[1,9] := MATRIX_STRUCTURE_NON_RETAIN.MATRIX_INT[1,7];

    MATRIX_STRUCTURE_NON_RETAIN.MATRIX_INT[2,0] := MATRIX_STRUCTURE_NON_RETAIN.MATRIX_INT[2,0] + 1;
    MATRIX_STRUCTURE_NON_RETAIN.MATRIX_INT[2,1] := MATRIX_STRUCTURE_NON_RETAIN.MATRIX_INT[2,1] + 1;
    MATRIX_STRUCTURE_NON_RETAIN.MATRIX_INT[2,2] := MATRIX_STRUCTURE_NON_RETAIN.MATRIX_INT[2,2] + 1;
    MATRIX_STRUCTURE_NON_RETAIN.MATRIX_INT[2,3] := MATRIX_STRUCTURE_NON_RETAIN.MATRIX_INT[2,3] + 1;
    MATRIX_STRUCTURE_NON_RETAIN.MATRIX_INT[2,4] := MATRIX_STRUCTURE_NON_RETAIN.MATRIX_INT[2,4] + 1;
    MATRIX_STRUCTURE_NON_RETAIN.MATRIX_INT[2,5] := MATRIX_STRUCTURE_NON_RETAIN.MATRIX_INT[2,5] + 1;
    MATRIX_STRUCTURE_NON_RETAIN.MATRIX_INT[2,6] := MATRIX_STRUCTURE_NON_RETAIN.MATRIX_INT[2,6] + 1;
    MATRIX_STRUCTURE_NON_RETAIN.MATRIX_INT[2,7] := MATRIX_STRUCTURE_NON_RETAIN.MATRIX_INT[2,7] + 1;
    MATRIX_STRUCTURE_NON_RETAIN.MATRIX_INT[2,8] := MATRIX_STRUCTURE_NON_RETAIN.MATRIX_INT[2,8] + 1;
    MATRIX_STRUCTURE_NON_RETAIN.MATRIX_INT[2,9] := MATRIX_STRUCTURE_NON_RETAIN.MATRIX_INT[2,9] + 1;

    MATRIX_STRUCTURE_NON_RETAIN.MATRIX_INT[3,0] := MATRIX_STRUCTURE_NON_RETAIN.MATRIX_INT[3,0] + 1;
    MATRIX_STRUCTURE_NON_RETAIN.MATRIX_INT[3,1] := MATRIX_STRUCTURE_NON_RETAIN.MATRIX_INT[3,1] + 1;
    MATRIX_STRUCTURE_NON_RETAIN.MATRIX_INT[3,2] := MATRIX_STRUCTURE_NON_RETAIN.MATRIX_INT[3,2] + 1;
    MATRIX_STRUCTURE_NON_RETAIN.MATRIX_INT[3,3] := MATRIX_STRUCTURE_NON_RETAIN.MATRIX_INT[3,3] + 1;
    MATRIX_STRUCTURE_NON_RETAIN.MATRIX_INT[3,4] := MATRIX_STRUCTURE_NON_RETAIN.MATRIX_INT[3,4] + 1;
    MATRIX_STRUCTURE_NON_RETAIN.MATRIX_INT[3,5] := MATRIX_STRUCTURE_NON_RETAIN.MATRIX_INT[3,5] + 1;
    MATRIX_STRUCTURE_NON_RETAIN.MATRIX_INT[3,6] := MATRIX_STRUCTURE_NON_RETAIN.MATRIX_INT[3,6] + 1;
    MATRIX_STRUCTURE_NON_RETAIN.MATRIX_INT[3,7] := MATRIX_STRUCTURE_NON_RETAIN.MATRIX_INT[3,7] + 1;
    MATRIX_STRUCTURE_NON_RETAIN.MATRIX_INT[3,8] := MATRIX_STRUCTURE_NON_RETAIN.MATRIX_INT[3,8] + 1;
    MATRIX_STRUCTURE_NON_RETAIN.MATRIX_INT[3,9] := MATRIX_STRUCTURE_NON_RETAIN.MATRIX_INT[3,9] + 1;

    MATRIX_STRUCTURE_NON_RETAIN.MATRIX_INT[4,0] := MATRIX_STRUCTURE_NON_RETAIN.MATRIX_INT[4,0] + 1;
    MATRIX_STRUCTURE_NON_RETAIN.MATRIX_INT[4,1] := MATRIX_STRUCTURE_NON_RETAIN.MATRIX_INT[4,1] + 1;
    MATRIX_STRUCTURE_NON_RETAIN.MATRIX_INT[4,2] := MATRIX_STRUCTURE_NON_RETAIN.MATRIX_INT[4,2] + 1;
    MATRIX_STRUCTURE_NON_RETAIN.MATRIX_INT[4,3] := MATRIX_STRUCTURE_NON_RETAIN.MATRIX_INT[4,3] + 1;
    MATRIX_STRUCTURE_NON_RETAIN.MATRIX_INT[4,4] := MATRIX_STRUCTURE_NON_RETAIN.MATRIX_INT[4,4] + 1;
    MATRIX_STRUCTURE_NON_RETAIN.MATRIX_INT[4,5] := MATRIX_STRUCTURE_NON_RETAIN.MATRIX_INT[4,5] + 1;
    MATRIX_STRUCTURE_NON_RETAIN.MATRIX_INT[4,6] := MATRIX_STRUCTURE_NON_RETAIN.MATRIX_INT[4,6] + 1;
    MATRIX_STRUCTURE_NON_RETAIN.MATRIX_INT[4,7] := MATRIX_STRUCTURE_NON_RETAIN.MATRIX_INT[4,7] + 1;
    MATRIX_STRUCTURE_NON_RETAIN.MATRIX_INT[4,8] := MATRIX_STRUCTURE_NON_RETAIN.MATRIX_INT[4,8] + 1;
    MATRIX_STRUCTURE_NON_RETAIN.MATRIX_INT[4,9] := MATRIX_STRUCTURE_NON_RETAIN.MATRIX_INT[4,9] + 1;

    MATRIX_STRUCTURE_NON_RETAIN.MATRIX_INT[5,0] := MATRIX_STRUCTURE_NON_RETAIN.MATRIX_INT[5,0] + 1;
    MATRIX_STRUCTURE_NON_RETAIN.MATRIX_INT[5,1] := MATRIX_STRUCTURE_NON_RETAIN.MATRIX_INT[5,1] + 1;
    MATRIX_STRUCTURE_NON_RETAIN.MATRIX_INT[5,2] := MATRIX_STRUCTURE_NON_RETAIN.MATRIX_INT[5,2] + 1;
    MATRIX_STRUCTURE_NON_RETAIN.MATRIX_INT[5,3] := MATRIX_STRUCTURE_NON_RETAIN.MATRIX_INT[5,3] + 1;
    MATRIX_STRUCTURE_NON_RETAIN.MATRIX_INT[5,4] := MATRIX_STRUCTURE_NON_RETAIN.MATRIX_INT[5,4] + 1;
    MATRIX_STRUCTURE_NON_RETAIN.MATRIX_INT[5,5] := MATRIX_STRUCTURE_NON_RETAIN.MATRIX_INT[5,5] + 1;
    MATRIX_STRUCTURE_NON_RETAIN.MATRIX_INT[5,6] := MATRIX_STRUCTURE_NON_RETAIN.MATRIX_INT[5,6] + 1;
    MATRIX_STRUCTURE_NON_RETAIN.MATRIX_INT[5,7] := MATRIX_STRUCTURE_NON_RETAIN.MATRIX_INT[5,7] + 1;
    MATRIX_STRUCTURE_NON_RETAIN.MATRIX_INT[5,8] := MATRIX_STRUCTURE_NON_RETAIN.MATRIX_INT[5,8] + 1;
    MATRIX_STRUCTURE_NON_RETAIN.MATRIX_INT[5,9] := MATRIX_STRUCTURE_NON_RETAIN.MATRIX_INT[5,9] + 1;
